    |   movel([0.182461, -1.429621, -2.539510, -0.743258, 1.570796, 1.753257],accel_mss,speed_ms,0,blend_radius_m)
    |   movel([0.183810, -1.429810, -2.539363, -0.743216, 1.570796, 1.754607],accel_mss,speed_ms,0,blend_radius_m)
    |   movel([0.185034, -1.430194, -2.539064, -0.743131, 1.570796, 1.755830],accel_mss,speed_ms,0,blend_radius_m)
    |   movel([0.186110, -1.430760, -2.538624, -0.743005, 1.570796, 1.756906],accel_mss,speed_ms,0,blend_radius_m)
    |   movel([0.187012, -1.431499, -2.538048, -0.742842, 1.570796, 1.757809],accel_mss,speed_ms,0,blend_radius_m)
    |   movel([0.187715, -1.432399, -2.537345, -0.742645, 1.570796, 1.758511],accel_mss,speed_ms,0,blend_radius_m)
    |   movel([0.188198, -1.433447, -2.536525, -0.742416, 1.570796, 1.758995],accel_mss,speed_ms,0,blend_radius_m)
    |   speed_ms = 0.005
    |   movel([0.188198, -1.425059, -2.532761, -0.754569, 1.570796, 1.758995],accel_mss,speed_ms,0,blend_radius_m)
    |   speed_ms = 0.040
    |   movel([0.160347, -1.408053, -2.545687, -0.758649, 1.570796, 1.731144],accel_mss,speed_ms,0,blend_radius_m)
    |   speed_ms = 0.005
    |   movel([0.160347, -1.416570, -2.549523, -0.746297, 1.570796, 1.731144],accel_mss,speed_ms,0,blend_radius_m)
    |   speed_ms = 0.025
    |   movel([0.161048, -1.416837, -2.549320, -0.746232, 1.570796, 1.731844],accel_mss,speed_ms,0,blend_radius_m)
    |   movel([0.161576, -1.417274, -2.548989, -0.746126, 1.570796, 1.732372],accel_mss,speed_ms,0,blend_radius_m)
    |   movel([0.161701, -1.417602, -2.548740, -0.746047, 1.570796, 1.732497],accel_mss,speed_ms,0,blend_radius_m)
    |   movel([0.161690, -1.417989, -2.548446, -0.745954, 1.570796, 1.732487],accel_mss,speed_ms,0,blend_radius_m)
    |   movel([0.161538, -1.418393, -2.548139, -0.745857, 1.570796, 1.732334],accel_mss,speed_ms,0,blend_radius_m)
    |   movel([0.161230, -1.418767, -2.547855, -0.745767, 1.570796, 1.732027],accel_mss,speed_ms,0,blend_radius_m)
    |   movel([0.160492, -1.419336, -2.547422, -0.745631, 1.570796, 1.731288],accel_mss,speed_ms,0,blend_radius_m)
    |   movel([0.160242, -1.419699, -2.547145, -0.745545, 1.570796, 1.731038],accel_mss,speed_ms,0,blend_radius_m)
    |   movel([0.160152, -1.420075, -2.546859, -0.745456, 1.570796, 1.730949],accel_mss,speed_ms,0,blend_radius_m)
    |   movel([0.160302, -1.420762, -2.546335, -0.745293, 1.570796, 1.731098],accel_mss,speed_ms,0,blend_radius_m)
    |   movel([0.160720, -1.421423, -2.545829, -0.745137, 1.570796, 1.731517],accel_mss,speed_ms,0,blend_radius_m)
    |   movel([0.161277, -1.421975, -2.545406, -0.745007, 1.570796, 1.732073],accel_mss,speed_ms,0,blend_radius_m)
    |   movel([0.161958, -1.422414, -2.545071, -0.744905, 1.570796, 1.732754],accel_mss,speed_ms,0,blend_radius_m)
    |   movel([0.162749, -1.422724, -2.544833, -0.744832, 1.570796, 1.733545],accel_mss,speed_ms,0,blend_radius_m)
    |   movel([0.162178, -1.423539, -2.544208, -0.744642, 1.570796, 1.732975],accel_mss,speed_ms,0,blend_radius_m)
    |   movel([0.161765, -1.424363, -2.543574, -0.744451, 1.570796, 1.732562],accel_mss,speed_ms,0,blend_radius_m)
    |   movel([0.161491, -1.425192, -2.542936, -0.744261, 1.570796, 1.732287],accel_mss,speed_ms,0,blend_radius_m)
    |   movel([0.161335, -1.426018, -2.542300, -0.744072, 1.570796, 1.732131],accel_mss,speed_ms,0,blend_radius_m)
    |   movel([0.161310, -1.427628, -2.541056, -0.743706, 1.570796, 1.732106],accel_mss,speed_ms,0,blend_radius_m)
    |   movel([0.161552, -1.429136, -2.539887, -0.743367, 1.570796, 1.732348],accel_mss,speed_ms,0,blend_radius_m)
    |   movel([0.161818, -1.430578, -2.538765, -0.743046, 1.570796, 1.732614],accel_mss,speed_ms,0,blend_radius_m)
    |   movel([0.161818, -1.431340, -2.538172, -0.742877, 1.570796, 1.732614],accel_mss,speed_ms,0,blend_radius_m)
    |   movel([0.161643, -1.432142, -2.537546, -0.742701, 1.570796, 1.732440],accel_mss,speed_ms,0,blend_radius_m)
    |   movel([0.161209, -1.432975, -2.536895, -0.742519, 1.570796, 1.732006],accel_mss,speed_ms,0,blend_radius_m)
    |   movel([0.160534, -1.433740, -2.536296, -0.742353, 1.570796, 1.731330],accel_mss,speed_ms,0,blend_radius_m)
    |   movel([0.159706, -1.434315, -2.535846, -0.742229, 1.570796, 1.730503],accel_mss,speed_ms,0,blend_radius_m)
    |   movel([0.158821, -1.434572, -2.535644, -0.742173, 1.570796, 1.729617],accel_mss,speed_ms,0,blend_radius_m)
    |   movel([0.159210, -1.435121, -2.535213, -0.742055, 1.570796, 1.730006],accel_mss,speed_ms,0,blend_radius_m)
    |   movel([0.159647, -1.436428, -2.534185, -0.741776, 1.570796, 1.730443],accel_mss,speed_ms,0,blend_radius_m)
    |   movel([0.159693, -1.437162, -2.533607, -0.741620, 1.570796, 1.730489],accel_mss,speed_ms,0,blend_radius_m)
    |   movel([0.159449, -1.438725, -2.532372, -0.741291, 1.570796, 1.730245],accel_mss,speed_ms,0,blend_radius_m)
    |   movel([0.159158, -1.439530, -2.531736, -0.741124, 1.570796, 1.729954],accel_mss,speed_ms,0,blend_radius_m)
    |   movel([0.158753, -1.440335, -2.531097, -0.740957, 1.570796, 1.729550],accel_mss,speed_ms,0,blend_radius_m)
    |   speed_ms = 0.005
    |   movel([0.158753, -1.432000, -2.527362, -0.753027, 1.570796, 1.729550],accel_mss,speed_ms,0,blend_radius_m)
    |   speed_ms = 0.040
    |   movel([0.154357, -1.432582, -2.526906, -0.752901, 1.570796, 1.725154],accel_mss,speed_ms,0,blend_radius_m)
    |   speed_ms = 0.005
    |   movel([0.154357, -1.440913, -2.530638, -0.740838, 1.570796, 1.725154],accel_mss,speed_ms,0,blend_radius_m)
    |   speed_ms = 0.025
    |   movel([0.157061, -1.447582, -2.525307, -0.739499, 1.570796, 1.727858],accel_mss,speed_ms,0,blend_radius_m)
    |   movel([0.157277, -1.448453, -2.524606, -0.739330, 1.570796, 1.728073],accel_mss,speed_ms,0,blend_radius_m)
    |   movel([0.157213, -1.448926, -2.524225, -0.739238, 1.570796, 1.728009],accel_mss,speed_ms,0,blend_radius_m)
    |   movel([0.156951, -1.449404, -2.523839, -0.739146, 1.570796, 1.727748],accel_mss,speed_ms,0,blend_radius_m)
    |   movel([0.156049, -1.450346, -2.523078, -0.738965, 1.570796, 1.726845],accel_mss,speed_ms,0,blend_radius_m)
    |   movel([0.155895, -1.450870, -2.522654, -0.738865, 1.570796, 1.726691],accel_mss,speed_ms,0,blend_radius_m)
    |   movel([0.155988, -1.451343, -2.522271, -0.738775, 1.570796, 1.726784],accel_mss,speed_ms,0,blend_radius_m)
    |   movel([0.156429, -1.451974, -2.521759, -0.738655, 1.570796, 1.727225],accel_mss,speed_ms,0,blend_radius_m)
    |   movel([0.157105, -1.452459, -2.521366, -0.738564, 1.570796, 1.727901],accel_mss,speed_ms,0,blend_radius_m)
    |   movel([0.158587, -1.453259, -2.520716, -0.738414, 1.570796, 1.729384],accel_mss,speed_ms,0,blend_radius_m)
    |   movel([0.159389, -1.453953, -2.520151, -0.738285, 1.570796, 1.730186],accel_mss,speed_ms,0,blend_radius_m)
    |   movel([0.160307, -1.455102, -2.519215, -0.738073, 1.570796, 1.731103],accel_mss,speed_ms,0,blend_radius_m)
    |   movel([0.160572, -1.455706, -2.518721, -0.737962, 1.570796, 1.731368],accel_mss,speed_ms,0,blend_radius_m)
    |   movel([0.160588, -1.456254, -2.518273, -0.737862, 1.570796, 1.731385],accel_mss,speed_ms,0,blend_radius_m)
    |   movel([0.160472, -1.456488, -2.518082, -0.737819, 1.570796, 1.731269],accel_mss,speed_ms,0,blend_radius_m)
    |   movel([0.160258, -1.456686, -2.517920, -0.737783, 1.570796, 1.731054],accel_mss,speed_ms,0,blend_radius_m)
    |   movel([0.159489, -1.456951, -2.517703, -0.737735, 1.570796, 1.730285],accel_mss,speed_ms,0,blend_radius_m)
    |   movel([0.159593, -1.457513, -2.517242, -0.737634, 1.570796, 1.730389],accel_mss,speed_ms,0,blend_radius_m)
    |   movel([0.159908, -1.458064, -2.516791, -0.737535, 1.570796, 1.730705],accel_mss,speed_ms,0,blend_radius_m)
    |   movel([0.160965, -1.459087, -2.515950, -0.737352, 1.570796, 1.731762],accel_mss,speed_ms,0,blend_radius_m)
    |   movel([0.163339, -1.460579, -2.514722, -0.737088, 1.570796, 1.734136],accel_mss,speed_ms,0,blend_radius_m)
    |   movel([0.164707, -1.461116, -2.514279, -0.736994, 1.570796, 1.735503],accel_mss,speed_ms,0,blend_radius_m)
    |   movel([0.166237, -1.461556, -2.513915, -0.736918, 1.570796, 1.737034],accel_mss,speed_ms,0,blend_radius_m)
    |   movel([0.167609, -1.462139, -2.513433, -0.736816, 1.570796, 1.738405],accel_mss,speed_ms,0,blend_radius_m)
    |   movel([0.168136, -1.462558, -2.513087, -0.736744, 1.570796, 1.738932],accel_mss,speed_ms,0,blend_radius_m)
    |   movel([0.168503, -1.463100, -2.512638, -0.736651, 1.570796, 1.739300],accel_mss,speed_ms,0,blend_radius_m)
    |   movel([0.168579, -1.463445, -2.512352, -0.736592, 1.570796, 1.739375],accel_mss,speed_ms,0,blend_radius_m)
    |   movel([0.168528, -1.463831, -2.512032, -0.736526, 1.570796, 1.739324],accel_mss,speed_ms,0,blend_radius_m)
    |   movel([0.168335, -1.464184, -2.511739, -0.736466, 1.570796, 1.739132],accel_mss,speed_ms,0,blend_radius_m)
    |   movel([0.167982, -1.464429, -2.511536, -0.736424, 1.570796, 1.738778],accel_mss,speed_ms,0,blend_radius_m)
    |   movel([0.167358, -1.464441, -2.511526, -0.736422, 1.570796, 1.738154],accel_mss,speed_ms,0,blend_radius_m)
    |   movel([0.164733, -1.463725, -2.512120, -0.736544, 1.570796, 1.735529],accel_mss,speed_ms,0,blend_radius_m)
    |   movel([0.162348, -1.462693, -2.512975, -0.736721, 1.570796, 1.733144],accel_mss,speed_ms,0,blend_radius_m)
    |   movel([0.162165, -1.463098, -2.512640, -0.736651, 1.570796, 1.732962],accel_mss,speed_ms,0,blend_radius_m)
    |   movel([0.162102, -1.463492, -2.512313, -0.736584, 1.570796, 1.732898],accel_mss,speed_ms,0,blend_radius_m)
    |   movel([0.162287, -1.464240, -2.511693, -0.736456, 1.570796, 1.733083],accel_mss,speed_ms,0,blend_radius_m)
    |   movel([0.162802, -1.464926, -2.511123, -0.736340, 1.570796, 1.733598],accel_mss,speed_ms,0,blend_radius_m)
    |   movel([0.163541, -1.465551, -2.510603, -0.736235, 1.570796, 1.734338],accel_mss,speed_ms,0,blend_radius_m)
    |   movel([0.165313, -1.466577, -2.509748, -0.736064, 1.570796, 1.736110],accel_mss,speed_ms,0,blend_radius_m)
    |   movel([0.166806, -1.467265, -2.509174, -0.735950, 1.570796, 1.737602],accel_mss,speed_ms,0,blend_radius_m)
    |   movel([0.167308, -1.467575, -2.508916, -0.735899, 1.570796, 1.738104],accel_mss,speed_ms,0,blend_radius_m)
    |   movel([0.167450, -1.467798, -2.508729, -0.735862, 1.570796, 1.738246],accel_mss,speed_ms,0,blend_radius_m)
    |   movel([0.167453, -1.468085, -2.508489, -0.735815, 1.570796, 1.738249],accel_mss,speed_ms,0,blend_radius_m)
    |   movel([0.167296, -1.468415, -2.508213, -0.735761, 1.570796, 1.738092],accel_mss,speed_ms,0,blend_radius_m)
    |   movel([0.167062, -1.468632, -2.508031, -0.735726, 1.570796, 1.737858],accel_mss,speed_ms,0,blend_radius_m)
    |   movel([0.166454, -1.468850, -2.507849, -0.735690, 1.570796, 1.737251],accel_mss,speed_ms,0,blend_radius_m)
    |   movel([0.165595, -1.469078, -2.507658, -0.735653, 1.570796, 1.736392],accel_mss,speed_ms,0,blend_radius_m)
    |   movel([0.165427, -1.469247, -2.507517, -0.735626, 1.570796, 1.736223],accel_mss,speed_ms,0,blend_radius_m)
    |   movel([0.165345, -1.469528, -2.507281, -0.735580, 1.570796, 1.736141],accel_mss,speed_ms,0,blend_radius_m)
    |   movel([0.165401, -1.469808, -2.507046, -0.735535, 1.570796, 1.736198],accel_mss,speed_ms,0,blend_radius_m)
    |   movel([0.165799, -1.470337, -2.506602, -0.735450, 1.570796, 1.736596],accel_mss,speed_ms,0,blend_radius_m)
    |   movel([0.166817, -1.471128, -2.505937, -0.735324, 1.570796, 1.737614],accel_mss,speed_ms,0,blend_radius_m)
    |   movel([0.171507, -1.474123, -2.503412, -0.734854, 1.570796, 1.742303],accel_mss,speed_ms,0,blend_radius_m)
    |   movel([0.171909, -1.474489, -2.503102, -0.734798, 1.570796, 1.742705],accel_mss,speed_ms,0,blend_radius_m)
    |   movel([0.172183, -1.474947, -2.502714, -0.734728, 1.570796, 1.742980],accel_mss,speed_ms,0,blend_radius_m)
    |   movel([0.172221, -1.475464, -2.502276, -0.734649, 1.570796, 1.743018],accel_mss,speed_ms,0,blend_radius_m)
    |   movel([0.171913, -1.476002, -2.501820, -0.734567, 1.570796, 1.742709],accel_mss,speed_ms,0,blend_radius_m)
    |   movel([0.171372, -1.476368, -2.501509, -0.734512, 1.570796, 1.742169],accel_mss,speed_ms,0,blend_radius_m)
    |   movel([0.170763, -1.476499, -2.501398, -0.734492, 1.570796, 1.741560],accel_mss,speed_ms,0,blend_radius_m)
    |   movel([0.170150, -1.476458, -2.501433, -0.734498, 1.570796, 1.740946],accel_mss,speed_ms,0,blend_radius_m)
    |   movel([0.169597, -1.476313, -2.501556, -0.734520, 1.570796, 1.740393],accel_mss,speed_ms,0,blend_radius_m)
    |   movel([0.166572, -1.475142, -2.502549, -0.734698, 1.570796, 1.737369],accel_mss,speed_ms,0,blend_radius_m)
    |   movel([0.163666, -1.473823, -2.503665, -0.734901, 1.570796, 1.734463],accel_mss,speed_ms,0,blend_radius_m)
    |   movel([0.160882, -1.472356, -2.504903, -0.735130, 1.570796, 1.731678],accel_mss,speed_ms,0,blend_radius_m)
    |   movel([0.158230, -1.470742, -2.506262, -0.735385, 1.570796, 1.729026],accel_mss,speed_ms,0,blend_radius_m)
    |   movel([0.157306, -1.470085, -2.506813, -0.735490, 1.570796, 1.728103],accel_mss,speed_ms,0,blend_radius_m)
    |   movel([0.156559, -1.469281, -2.507488, -0.735620, 1.570796, 1.727356],accel_mss,speed_ms,0,blend_radius_m)
    |   movel([0.156265, -1.468703, -2.507972, -0.735714, 1.570796, 1.727061],accel_mss,speed_ms,0,blend_radius_m)
    |   movel([0.156066, -1.468071, -2.508501, -0.735817, 1.570796, 1.726862],accel_mss,speed_ms,0,blend_radius_m)
    |   movel([0.155838, -1.466713, -2.509635, -0.736041, 1.570796, 1.726634],accel_mss,speed_ms,0,blend_radius_m)
    |   movel([0.155601, -1.461616, -2.513866, -0.736907, 1.570796, 1.726397],accel_mss,speed_ms,0,blend_radius_m)
    |   movel([0.155370, -1.460235, -2.515006, -0.737149, 1.570796, 1.726167],accel_mss,speed_ms,0,blend_radius_m)
    |   movel([0.154966, -1.459071, -2.515963, -0.737355, 1.570796, 1.725762],accel_mss,speed_ms,0,blend_radius_m)
    |   movel([0.154681, -1.458614, -2.516339, -0.737436, 1.570796, 1.725477],accel_mss,speed_ms,0,blend_radius_m)
    |   movel([0.154331, -1.458258, -2.516631, -0.737500, 1.570796, 1.725127],accel_mss,speed_ms,0,blend_radius_m)
    |   movel([0.153911, -1.458025, -2.516822, -0.737541, 1.570796, 1.724707],accel_mss,speed_ms,0,blend_radius_m)
    |   movel([0.153414, -1.457927, -2.516903, -0.737559, 1.570796, 1.724210],accel_mss,speed_ms,0,blend_radius_m)
    |   movel([0.152456, -1.457979, -2.516860, -0.737550, 1.570796, 1.723252],accel_mss,speed_ms,0,blend_radius_m)
    |   movel([0.152013, -1.457959, -2.516877, -0.737553, 1.570796, 1.722809],accel_mss,speed_ms,0,blend_radius_m)
    |   movel([0.151669, -1.457806, -2.517002, -0.737581, 1.570796, 1.722466],accel_mss,speed_ms,0,blend_radius_m)
    |   movel([0.151472, -1.457323, -2.517398, -0.737668, 1.570796, 1.722268],accel_mss,speed_ms,0,blend_radius_m)
    |   movel([0.151536, -1.456708, -2.517902, -0.737779, 1.570796, 1.722333],accel_mss,speed_ms,0,blend_radius_m)
    |   movel([0.151846, -1.454712, -2.519533, -0.738144, 1.570796, 1.722643],accel_mss,speed_ms,0,blend_radius_m)
    |   movel([0.152006, -1.452762, -2.521120, -0.738507, 1.570796, 1.722802],accel_mss,speed_ms,0,blend_radius_m)
    |   movel([0.151950, -1.448972, -2.524188, -0.739229, 1.570796, 1.722746],accel_mss,speed_ms,0,blend_radius_m)
    |   movel([0.151537, -1.445268, -2.527165, -0.739956, 1.570796, 1.722334],accel_mss,speed_ms,0,blend_radius_m)
    |   movel([0.150932, -1.441582, -2.530107, -0.740700, 1.570796, 1.721728],accel_mss,speed_ms,0,blend_radius_m)
    |   speed_ms = 0.005
    |   movel([0.150932, -1.433257, -2.526377, -0.752755, 1.570796, 1.721728],accel_mss,speed_ms,0,blend_radius_m)
    |   speed_ms = 0.040
    |   movel([0.148558, -1.439611, -2.521359, -0.751419, 1.570796, 1.719355],accel_mss,speed_ms,0,blend_radius_m)
    |   speed_ms = 0.005
    |   movel([0.148558, -1.447887, -2.525062, -0.739440, 1.570796, 1.719355],accel_mss,speed_ms,0,blend_radius_m)
    |   speed_ms = 0.025
    |   movel([0.147293, -1.452117, -2.521643, -0.738628, 1.570796, 1.718089],accel_mss,speed_ms,0,blend_radius_m)
    |   movel([0.146519, -1.454236, -2.519921, -0.738232, 1.570796, 1.717315],accel_mss,speed_ms,0,blend_radius_m)
    |   movel([0.145655, -1.456350, -2.518195, -0.737844, 1.570796, 1.716451],accel_mss,speed_ms,0,blend_radius_m)
    |   movel([0.144468, -1.455618, -2.518793, -0.737978, 1.570796, 1.715264],accel_mss,speed_ms,0,blend_radius_m)
    |   movel([0.144245, -1.455516, -2.518877, -0.737997, 1.570796, 1.715041],accel_mss,speed_ms,0,blend_radius_m)
    |   movel([0.143973, -1.455537, -2.518860, -0.737993, 1.570796, 1.714769],accel_mss,speed_ms,0,blend_radius_m)
    |   movel([0.143715, -1.455735, -2.518697, -0.737956, 1.570796, 1.714512],accel_mss,speed_ms,0,blend_radius_m)
    |   movel([0.143536, -1.456005, -2.518477, -0.737907, 1.570796, 1.714332],accel_mss,speed_ms,0,blend_radius_m)
    |   movel([0.142423, -1.457670, -2.517114, -0.737605, 1.570796, 1.713219],accel_mss,speed_ms,0,blend_radius_m)
    |   movel([0.141061, -1.459243, -2.515822, -0.737324, 1.570796, 1.711857],accel_mss,speed_ms,0,blend_radius_m)
    |   movel([0.140683, -1.459568, -2.515554, -0.737266, 1.570796, 1.711479],accel_mss,speed_ms,0,blend_radius_m)
    |   movel([0.140276, -1.459709, -2.515438, -0.737242, 1.570796, 1.711073],accel_mss,speed_ms,0,blend_radius_m)
    |   movel([0.140039, -1.459566, -2.515556, -0.737267, 1.570796, 1.710835],accel_mss,speed_ms,0,blend_radius_m)
    |   movel([0.139948, -1.459290, -2.515783, -0.737316, 1.570796, 1.710744],accel_mss,speed_ms,0,blend_radius_m)
    |   movel([0.139802, -1.457440, -2.517302, -0.737647, 1.570796, 1.710598],accel_mss,speed_ms,0,blend_radius_m)
    |   movel([0.140013, -1.455473, -2.518911, -0.738004, 1.570796, 1.710809],accel_mss,speed_ms,0,blend_radius_m)
    |   speed_ms = 0.005
    |   movel([0.140013, -1.447256, -2.515240, -0.749893, 1.570796, 1.710809],accel_mss,speed_ms,0,blend_radius_m)
    |   speed_ms = 0.040
    |   movel([0.143541, -1.450689, -2.512464, -0.749236, 1.570796, 1.714337],accel_mss,speed_ms,0,blend_radius_m)
    |   speed_ms = 0.005
    |   movel([0.143541, -1.458879, -2.516121, -0.737389, 1.570796, 1.714337],accel_mss,speed_ms,0,blend_radius_m)
    |   speed_ms = 0.025
    |   movel([0.143262, -1.461761, -2.513746, -0.736882, 1.570796, 1.714058],accel_mss,speed_ms,0,blend_radius_m)
    |   movel([0.142955, -1.463237, -2.512525, -0.736627, 1.570796, 1.713751],accel_mss,speed_ms,0,blend_radius_m)
    |   movel([0.142021, -1.466218, -2.510047, -0.736123, 1.570796, 1.712817],accel_mss,speed_ms,0,blend_radius_m)
    |   movel([0.141397, -1.467713, -2.508800, -0.735876, 1.570796, 1.712194],accel_mss,speed_ms,0,blend_radius_m)
    |   movel([0.139852, -1.470677, -2.506317, -0.735396, 1.570796, 1.710648],accel_mss,speed_ms,0,blend_radius_m)
    |   movel([0.140038, -1.469700, -2.507136, -0.735552, 1.570796, 1.710834],accel_mss,speed_ms,0,blend_radius_m)
    |   movel([0.139919, -1.468812, -2.507881, -0.735696, 1.570796, 1.710715],accel_mss,speed_ms,0,blend_radius_m)
    |   movel([0.139512, -1.468072, -2.508500, -0.735817, 1.570796, 1.710308],accel_mss,speed_ms,0,blend_radius_m)
    |   movel([0.138834, -1.467542, -2.508943, -0.735904, 1.570796, 1.709630],accel_mss,speed_ms,0,blend_radius_m)
    |   speed_ms = 0.005
    |   movel([0.138834, -1.459420, -2.505321, -0.747648, 1.570796, 1.709630],accel_mss,speed_ms,0,blend_radius_m)
    |   speed_ms = 0.040
    |   movel([0.126690, -1.463689, -2.501786, -0.746913, 1.570796, 1.697487],accel_mss,speed_ms,0,blend_radius_m)
    |   speed_ms = 0.005
    |   movel([0.126690, -1.471777, -2.505391, -0.735221, 1.570796, 1.697487],accel_mss,speed_ms,0,blend_radius_m)
    |   speed_ms = 0.025
    |   movel([0.124728, -1.473662, -2.503801, -0.734926, 1.570796, 1.695524],accel_mss,speed_ms,0,blend_radius_m)
    |   movel([0.122583, -1.475378, -2.502349, -0.734662, 1.570796, 1.693379],accel_mss,speed_ms,0,blend_radius_m)
    |   movel([0.120295, -1.476899, -2.501058, -0.734432, 1.570796, 1.691091],accel_mss,speed_ms,0,blend_radius_m)
    |   movel([0.117902, -1.478198, -2.499953, -0.734238, 1.570796, 1.688698],accel_mss,speed_ms,0,blend_radius_m)
    |   movel([0.118428, -1.477273, -2.500740, -0.734376, 1.570796, 1.689224],accel_mss,speed_ms,0,blend_radius_m)
    |   movel([0.118796, -1.476390, -2.501491, -0.734509, 1.570796, 1.689592],accel_mss,speed_ms,0,blend_radius_m)
    |   movel([0.118980, -1.475627, -2.502138, -0.734624, 1.570796, 1.689777],accel_mss,speed_ms,0,blend_radius_m)
    |   movel([0.118959, -1.475064, -2.502615, -0.734710, 1.570796, 1.689756],accel_mss,speed_ms,0,blend_radius_m)
    |   movel([0.118706, -1.474786, -2.502850, -0.734752, 1.570796, 1.689502],accel_mss,speed_ms,0,blend_radius_m)
    |   movel([0.118486, -1.474778, -2.502857, -0.734754, 1.570796, 1.689283],accel_mss,speed_ms,0,blend_radius_m)
    |   movel([0.118196, -1.474870, -2.502779, -0.734740, 1.570796, 1.688992],accel_mss,speed_ms,0,blend_radius_m)
    |   movel([0.117408, -1.475399, -2.502331, -0.734659, 1.570796, 1.688204],accel_mss,speed_ms,0,blend_radius_m)
    |   movel([0.115476, -1.477294, -2.500723, -0.734373, 1.570796, 1.686272],accel_mss,speed_ms,0,blend_radius_m)
    |   movel([0.114562, -1.478102, -2.500034, -0.734253, 1.570796, 1.685358],accel_mss,speed_ms,0,blend_radius_m)
    |   movel([0.112567, -1.479569, -2.498783, -0.734037, 1.570796, 1.683364],accel_mss,speed_ms,0,blend_radius_m)
    |   movel([0.111510, -1.480208, -2.498237, -0.733944, 1.570796, 1.682306],accel_mss,speed_ms,0,blend_radius_m)
    |   movel([0.110428, -1.480767, -2.497759, -0.733864, 1.570796, 1.681224],accel_mss,speed_ms,0,blend_radius_m)
    |   movel([0.109332, -1.481239, -2.497354, -0.733796, 1.570796, 1.680128],accel_mss,speed_ms,0,blend_radius_m)
    |   movel([0.108237, -1.481609, -2.497037, -0.733743, 1.570796, 1.679033],accel_mss,speed_ms,0,blend_radius_m)
    |   movel([0.109495, -1.480213, -2.498233, -0.733944, 1.570796, 1.680291],accel_mss,speed_ms,0,blend_radius_m)
    |   movel([0.110712, -1.478790, -2.499448, -0.734151, 1.570796, 1.681508],accel_mss,speed_ms,0,blend_radius_m)
    |   movel([0.111231, -1.477810, -2.500283, -0.734296, 1.570796, 1.682028],accel_mss,speed_ms,0,blend_radius_m)
    |   movel([0.111476, -1.476835, -2.501112, -0.734442, 1.570796, 1.682273],accel_mss,speed_ms,0,blend_radius_m)
    |   movel([0.111406, -1.476498, -2.501399, -0.734492, 1.570796, 1.682202],accel_mss,speed_ms,0,blend_radius_m)
    |   movel([0.111156, -1.476339, -2.501534, -0.734516, 1.570796, 1.681952],accel_mss,speed_ms,0,blend_radius_m)
    |   movel([0.110695, -1.476418, -2.501466, -0.734504, 1.570796, 1.681491],accel_mss,speed_ms,0,blend_radius_m)
    |   movel([0.109985, -1.476796, -2.501145, -0.734447, 1.570796, 1.680781],accel_mss,speed_ms,0,blend_radius_m)
    |   movel([0.106293, -1.479270, -2.499038, -0.734081, 1.570796, 1.677090],accel_mss,speed_ms,0,blend_radius_m)
    |   movel([0.104413, -1.480308, -2.498151, -0.733930, 1.570796, 1.675210],accel_mss,speed_ms,0,blend_radius_m)
    |   movel([0.103458, -1.480699, -2.497817, -0.733873, 1.570796, 1.674254],accel_mss,speed_ms,0,blend_radius_m)
    |   movel([0.102487, -1.480974, -2.497581, -0.733834, 1.570796, 1.673283],accel_mss,speed_ms,0,blend_radius_m)
    |   speed_ms = 0.005
    |   movel([0.102487, -1.472960, -2.494014, -0.745416, 1.570796, 1.673283],accel_mss,speed_ms,0,blend_radius_m)
    |   speed_ms = 0.040
    |   movel([0.118652, -1.454320, -2.509507, -0.748562, 1.570796, 1.689448],accel_mss,speed_ms,0,blend_radius_m)
    |   speed_ms = 0.005
    |   movel([0.118652, -1.462482, -2.513150, -0.736757, 1.570796, 1.689448],accel_mss,speed_ms,0,blend_radius_m)
    |   speed_ms = 0.025
    |   movel([0.118575, -1.461266, -2.514155, -0.736968, 1.570796, 1.689372],accel_mss,speed_ms,0,blend_radius_m)
    |   movel([0.118788, -1.459980, -2.515216, -0.737194, 1.570796, 1.689584],accel_mss,speed_ms,0,blend_radius_m)
    |   movel([0.119258, -1.458648, -2.516311, -0.737430, 1.570796, 1.690055],accel_mss,speed_ms,0,blend_radius_m)
    |   movel([0.119955, -1.457301, -2.517416, -0.737672, 1.570796, 1.690752],accel_mss,speed_ms,0,blend_radius_m)
    |   movel([0.120854, -1.455963, -2.518511, -0.737915, 1.570796, 1.691651],accel_mss,speed_ms,0,blend_radius_m)
    |   movel([0.121920, -1.454666, -2.519570, -0.738153, 1.570796, 1.692717],accel_mss,speed_ms,0,blend_radius_m)
    |   movel([0.123128, -1.453435, -2.520573, -0.738381, 1.570796, 1.693924],accel_mss,speed_ms,0,blend_radius_m)
    |   movel([0.124442, -1.452300, -2.521495, -0.738594, 1.570796, 1.695239],accel_mss,speed_ms,0,blend_radius_m)
    |   movel([0.126164, -1.451030, -2.522525, -0.738834, 1.570796, 1.696960],accel_mss,speed_ms,0,blend_radius_m)
    |   movel([0.129687, -1.448583, -2.524501, -0.739304, 1.570796, 1.700483],accel_mss,speed_ms,0,blend_radius_m)
    |   movel([0.131359, -1.447249, -2.525575, -0.739565, 1.570796, 1.702155],accel_mss,speed_ms,0,blend_radius_m)
    |   movel([0.132860, -1.445714, -2.526807, -0.739867, 1.570796, 1.703657],accel_mss,speed_ms,0,blend_radius_m)
    |   movel([0.133496, -1.444883, -2.527473, -0.740033, 1.570796, 1.704293],accel_mss,speed_ms,0,blend_radius_m)
    |   movel([0.134024, -1.444034, -2.528152, -0.740203, 1.570796, 1.704821],accel_mss,speed_ms,0,blend_radius_m)
    |   movel([0.134421, -1.443187, -2.528828, -0.740374, 1.570796, 1.705217],accel_mss,speed_ms,0,blend_radius_m)
    |   movel([0.134665, -1.442360, -2.529488, -0.740542, 1.570796, 1.705461],accel_mss,speed_ms,0,blend_radius_m)
    |   movel([0.134728, -1.441575, -2.530112, -0.740702, 1.570796, 1.705524],accel_mss,speed_ms,0,blend_radius_m)
    |   movel([0.134585, -1.440854, -2.530685, -0.740850, 1.570796, 1.705381],accel_mss,speed_ms,0,blend_radius_m)
    |   speed_ms = 0.005
    |   movel([0.134585, -1.432523, -2.526953, -0.752914, 1.570796, 1.705381],accel_mss,speed_ms,0,blend_radius_m)
    |   speed_ms = 0.040
    |   movel([0.133004, -1.426801, -2.531413, -0.754175, 1.570796, 1.703800],accel_mss,speed_ms,0,blend_radius_m)
    |   speed_ms = 0.005
    |   movel([0.133004, -1.435175, -2.535170, -0.742043, 1.570796, 1.703800],accel_mss,speed_ms,0,blend_radius_m)
    |   speed_ms = 0.025
    |   movel([0.131954, -1.439890, -2.531450, -0.741049, 1.570796, 1.702750],accel_mss,speed_ms,0,blend_radius_m)
    |   movel([0.131474, -1.440949, -2.530610, -0.740830, 1.570796, 1.702271],accel_mss,speed_ms,0,blend_radius_m)
    |   movel([0.130669, -1.441933, -2.529828, -0.740629, 1.570796, 1.701465],accel_mss,speed_ms,0,blend_radius_m)
    |   movel([0.129641, -1.442790, -2.529145, -0.740454, 1.570796, 1.700437],accel_mss,speed_ms,0,blend_radius_m)
    |   movel([0.126104, -1.445221, -2.527202, -0.739965, 1.570796, 1.696900],accel_mss,speed_ms,0,blend_radius_m)
    |   movel([0.124928, -1.446193, -2.526423, -0.739773, 1.570796, 1.695724],accel_mss,speed_ms,0,blend_radius_m)
    |   movel([0.123829, -1.447231, -2.525590, -0.739568, 1.570796, 1.694626],accel_mss,speed_ms,0,blend_radius_m)
    |   movel([0.122817, -1.448321, -2.524713, -0.739355, 1.570796, 1.693613],accel_mss,speed_ms,0,blend_radius_m)
    |   movel([0.121989, -1.449445, -2.523806, -0.739138, 1.570796, 1.692785],accel_mss,speed_ms,0,blend_radius_m)
    |   movel([0.121311, -1.450605, -2.522869, -0.738915, 1.570796, 1.692107],accel_mss,speed_ms,0,blend_radius_m)
    |   movel([0.120646, -1.451760, -2.521933, -0.738696, 1.570796, 1.691443],accel_mss,speed_ms,0,blend_radius_m)
    |   movel([0.119860, -1.452874, -2.521028, -0.738486, 1.570796, 1.690656],accel_mss,speed_ms,0,blend_radius_m)
    |   movel([0.118748, -1.450438, -2.523003, -0.738947, 1.570796, 1.689544],accel_mss,speed_ms,0,blend_radius_m)
    |   movel([0.118765, -1.449672, -2.523623, -0.739094, 1.570796, 1.689562],accel_mss,speed_ms,0,blend_radius_m)
    |   movel([0.118930, -1.448892, -2.524253, -0.739245, 1.570796, 1.689726],accel_mss,speed_ms,0,blend_radius_m)
    |   movel([0.119240, -1.448096, -2.524894, -0.739399, 1.570796, 1.690036],accel_mss,speed_ms,0,blend_radius_m)
    |   movel([0.119703, -1.447279, -2.525552, -0.739559, 1.570796, 1.690499],accel_mss,speed_ms,0,blend_radius_m)
    |   movel([0.120629, -1.446199, -2.526419, -0.739771, 1.570796, 1.691425],accel_mss,speed_ms,0,blend_radius_m)
    |   movel([0.122024, -1.444944, -2.527424, -0.740021, 1.570796, 1.692820],accel_mss,speed_ms,0,blend_radius_m)
    |   movel([0.125487, -1.442187, -2.529625, -0.740577, 1.570796, 1.696284],accel_mss,speed_ms,0,blend_radius_m)
    |   movel([0.127192, -1.440827, -2.530706, -0.740855, 1.570796, 1.697988],accel_mss,speed_ms,0,blend_radius_m)
    |   movel([0.128630, -1.439573, -2.531701, -0.741115, 1.570796, 1.699426],accel_mss,speed_ms,0,blend_radius_m)
    |   movel([0.129616, -1.438498, -2.532552, -0.741339, 1.570796, 1.700412],accel_mss,speed_ms,0,blend_radius_m)
    |   movel([0.129882, -1.438049, -2.532907, -0.741433, 1.570796, 1.700679],accel_mss,speed_ms,0,blend_radius_m)
    |   movel([0.129964, -1.437670, -2.533206, -0.741513, 1.570796, 1.700761],accel_mss,speed_ms,0,blend_radius_m)
    |   speed_ms = 0.005
    |   movel([0.129964, -1.429314, -2.529460, -0.753615, 1.570796, 1.700761],accel_mss,speed_ms,0,blend_radius_m)
    |   speed_ms = 0.040
    |   movel([0.122893, -1.428717, -2.529925, -0.753747, 1.570796, 1.693690],accel_mss,speed_ms,0,blend_radius_m)
    |   speed_ms = 0.005
    |   movel([0.122893, -1.437077, -2.533674, -0.741638, 1.570796, 1.693690],accel_mss,speed_ms,0,blend_radius_m)
    |   speed_ms = 0.025
    |   movel([0.122209, -1.437007, -2.533729, -0.741653, 1.570796, 1.693006],accel_mss,speed_ms,0,blend_radius_m)
    |   movel([0.121626, -1.436800, -2.533892, -0.741697, 1.570796, 1.692422],accel_mss,speed_ms,0,blend_radius_m)
    |   movel([0.120719, -1.436071, -2.534466, -0.741852, 1.570796, 1.691516],accel_mss,speed_ms,0,blend_radius_m)
    |   movel([0.120087, -1.435054, -2.535266, -0.742070, 1.570796, 1.690884],accel_mss,speed_ms,0,blend_radius_m)
    |   movel([0.119648, -1.433912, -2.536162, -0.742316, 1.570796, 1.690444],accel_mss,speed_ms,0,blend_radius_m)
    |   movel([0.119577, -1.433458, -2.536517, -0.742414, 1.570796, 1.690374],accel_mss,speed_ms,0,blend_radius_m)
    |   movel([0.119940, -1.432671, -2.537133, -0.742585, 1.570796, 1.690736],accel_mss,speed_ms,0,blend_radius_m)
    |   movel([0.121281, -1.430471, -2.538849, -0.743069, 1.570796, 1.692078],accel_mss,speed_ms,0,blend_radius_m)
    |   movel([0.123710, -1.426009, -2.542307, -0.744074, 1.570796, 1.694506],accel_mss,speed_ms,0,blend_radius_m)
    |   movel([0.124792, -1.423757, -2.544040, -0.744592, 1.570796, 1.695589],accel_mss,speed_ms,0,blend_radius_m)
    |   speed_ms = 0.005
    |   movel([0.124792, -1.415295, -2.540235, -0.756859, 1.570796, 1.695589],accel_mss,speed_ms,0,blend_radius_m)
    |   speed_ms = 0.040
    |   movel([0.120439, -1.416998, -2.538942, -0.756450, 1.570796, 1.691236],accel_mss,speed_ms,0,blend_radius_m)
    |   speed_ms = 0.005
    |   movel([0.120439, -1.425447, -2.542740, -0.744202, 1.570796, 1.691236],accel_mss,speed_ms,0,blend_radius_m)
    |   speed_ms = 0.025
    |   movel([0.119935, -1.426809, -2.541688, -0.743891, 1.570796, 1.690731],accel_mss,speed_ms,0,blend_radius_m)
    |   movel([0.119253, -1.428166, -2.540638, -0.743584, 1.570796, 1.690049],accel_mss,speed_ms,0,blend_radius_m)
    |   movel([0.118343, -1.429439, -2.539651, -0.743299, 1.570796, 1.689139],accel_mss,speed_ms,0,blend_radius_m)
    |   movel([0.117785, -1.430022, -2.539198, -0.743169, 1.570796, 1.688582],accel_mss,speed_ms,0,blend_radius_m)
    |   movel([0.116540, -1.431083, -2.538372, -0.742934, 1.570796, 1.687336],accel_mss,speed_ms,0,blend_radius_m)
    |   movel([0.116272, -1.431628, -2.537947, -0.742814, 1.570796, 1.687068],accel_mss,speed_ms,0,blend_radius_m)
    |   movel([0.114788, -1.435842, -2.534646, -0.741901, 1.570796, 1.685584],accel_mss,speed_ms,0,blend_radius_m)
    |   movel([0.114658, -1.436249, -2.534326, -0.741814, 1.570796, 1.685455],accel_mss,speed_ms,0,blend_radius_m)
    |   movel([0.114654, -1.436620, -2.534034, -0.741735, 1.570796, 1.685450],accel_mss,speed_ms,0,blend_radius_m)
    |   movel([0.114992, -1.436970, -2.533758, -0.741661, 1.570796, 1.685789],accel_mss,speed_ms,0,blend_radius_m)
    |   movel([0.115542, -1.437129, -2.533633, -0.741627, 1.570796, 1.686338],accel_mss,speed_ms,0,blend_radius_m)
    |   movel([0.117152, -1.437524, -2.533321, -0.741544, 1.570796, 1.687949],accel_mss,speed_ms,0,blend_radius_m)
    |   movel([0.118641, -1.438082, -2.532881, -0.741426, 1.570796, 1.689437],accel_mss,speed_ms,0,blend_radius_m)
    |   movel([0.119908, -1.438862, -2.532264, -0.741263, 1.570796, 1.690705],accel_mss,speed_ms,0,blend_radius_m)
    |   movel([0.120845, -1.439931, -2.531417, -0.741040, 1.570796, 1.691642],accel_mss,speed_ms,0,blend_radius_m)
    |   speed_ms = 0.005
    |   movel([0.120845, -1.431593, -2.527681, -0.753115, 1.570796, 1.691642],accel_mss,speed_ms,0,blend_radius_m)
    |   speed_ms = 0.040
    |   movel([0.117067, -1.442493, -2.519063, -0.750834, 1.570796, 1.687863],accel_mss,speed_ms,0,blend_radius_m)
    |   speed_ms = 0.005
    |   movel([0.117067, -1.450747, -2.522754, -0.738888, 1.570796, 1.687863],accel_mss,speed_ms,0,blend_radius_m)
    |   speed_ms = 0.025
    |   movel([0.116755, -1.450955, -2.522585, -0.738849, 1.570796, 1.687552],accel_mss,speed_ms,0,blend_radius_m)
    |   movel([0.116482, -1.451240, -2.522354, -0.738794, 1.570796, 1.687279],accel_mss,speed_ms,0,blend_radius_m)
    |   movel([0.115440, -1.452783, -2.521102, -0.738503, 1.570796, 1.686236],accel_mss,speed_ms,0,blend_radius_m)
    |   movel([0.115251, -1.452911, -2.520998, -0.738479, 1.570796, 1.686047],accel_mss,speed_ms,0,blend_radius_m)
    |   movel([0.114957, -1.452931, -2.520983, -0.738476, 1.570796, 1.685753],accel_mss,speed_ms,0,blend_radius_m)
    |   movel([0.114717, -1.452784, -2.521102, -0.738503, 1.570796, 1.685513],accel_mss,speed_ms,0,blend_radius_m)
    |   movel([0.114388, -1.452168, -2.521602, -0.738619, 1.570796, 1.685184],accel_mss,speed_ms,0,blend_radius_m)
    |   movel([0.114191, -1.450864, -2.522659, -0.738866, 1.570796, 1.684987],accel_mss,speed_ms,0,blend_radius_m)
    |   movel([0.114441, -1.449533, -2.523735, -0.739121, 1.570796, 1.685237],accel_mss,speed_ms,0,blend_radius_m)
    |   movel([0.114918, -1.448160, -2.524842, -0.739387, 1.570796, 1.685715],accel_mss,speed_ms,0,blend_radius_m)
    |   movel([0.115514, -1.446802, -2.525935, -0.739652, 1.570796, 1.686310],accel_mss,speed_ms,0,blend_radius_m)
    |   movel([0.116247, -1.445501, -2.526978, -0.739910, 1.570796, 1.687043],accel_mss,speed_ms,0,blend_radius_m)
    |   movel([0.117110, -1.444258, -2.527973, -0.740158, 1.570796, 1.687906],accel_mss,speed_ms,0,blend_radius_m)
    |   movel([0.118098, -1.443071, -2.528921, -0.740397, 1.570796, 1.688895],accel_mss,speed_ms,0,blend_radius_m)
    |   movel([0.119208, -1.441937, -2.529825, -0.740628, 1.570796, 1.690004],accel_mss,speed_ms,0,blend_radius_m)
    |   movel([0.120429, -1.440856, -2.530683, -0.740849, 1.570796, 1.691225],accel_mss,speed_ms,0,blend_radius_m)
    |   movel([0.121760, -1.439825, -2.531502, -0.741063, 1.570796, 1.692556],accel_mss,speed_ms,0,blend_radius_m)
    |   movel([0.123193, -1.438843, -2.532279, -0.741267, 1.570796, 1.693989],accel_mss,speed_ms,0,blend_radius_m)
    |   movel([0.125150, -1.437339, -2.533467, -0.741583, 1.570796, 1.695946],accel_mss,speed_ms,0,blend_radius_m)
    |   movel([0.127154, -1.435515, -2.534903, -0.741971, 1.570796, 1.697951],accel_mss,speed_ms,0,blend_radius_m)
    |   movel([0.129283, -1.433367, -2.536588, -0.742434, 1.570796, 1.700079],accel_mss,speed_ms,0,blend_radius_m)
    |   speed_ms = 0.005
    |   movel([0.129283, -1.424978, -2.532824, -0.754587, 1.570796, 1.700079],accel_mss,speed_ms,0,blend_radius_m)
    |   speed_ms = 0.040
    |   movel([0.127232, -1.425091, -2.532736, -0.754561, 1.570796, 1.698028],accel_mss,speed_ms,0,blend_radius_m)
    |   speed_ms = 0.005
    |   movel([0.127232, -1.433479, -2.536500, -0.742409, 1.570796, 1.698028],accel_mss,speed_ms,0,blend_radius_m)
    |   speed_ms = 0.025
    |   movel([0.128714, -1.430246, -2.539024, -0.743119, 1.570796, 1.699510],accel_mss,speed_ms,0,blend_radius_m)
    |   movel([0.130407, -1.427011, -2.541533, -0.743845, 1.570796, 1.701204],accel_mss,speed_ms,0,blend_radius_m)
    |   movel([0.131385, -1.425421, -2.542760, -0.744208, 1.570796, 1.702181],accel_mss,speed_ms,0,blend_radius_m)
    |   movel([0.132470, -1.423864, -2.543958, -0.744567, 1.570796, 1.703266],accel_mss,speed_ms,0,blend_radius_m)
    |   movel([0.133689, -1.422351, -2.545118, -0.744919, 1.570796, 1.704486],accel_mss,speed_ms,0,blend_radius_m)
    |   movel([0.135054, -1.420898, -2.546230, -0.745261, 1.570796, 1.705850],accel_mss,speed_ms,0,blend_radius_m)
    |   movel([0.138900, -1.417385, -2.548904, -0.746099, 1.570796, 1.709697],accel_mss,speed_ms,0,blend_radius_m)
    |   movel([0.140533, -1.415752, -2.550142, -0.746496, 1.570796, 1.711330],accel_mss,speed_ms,0,blend_radius_m)
    |   movel([0.141287, -1.414895, -2.550789, -0.746705, 1.570796, 1.712083],accel_mss,speed_ms,0,blend_radius_m)
    |   movel([0.141949, -1.413997, -2.551466, -0.746926, 1.570796, 1.712745],accel_mss,speed_ms,0,blend_radius_m)
    |   movel([0.143293, -1.411156, -2.553601, -0.747632, 1.570796, 1.714090],accel_mss,speed_ms,0,blend_radius_m)
    |   speed_ms = 0.005
    |   movel([0.143293, -1.402599, -2.549742, -0.760049, 1.570796, 1.714090],accel_mss,speed_ms,0,blend_radius_m)
    |   speed_ms = 0.040
    |   movel([0.146560, -1.395993, -2.554595, -0.761802, 1.570796, 1.717356],accel_mss,speed_ms,0,blend_radius_m)
    |   speed_ms = 0.005
    |   movel([0.146560, -1.404599, -2.558482, -0.749308, 1.570796, 1.717356],accel_mss,speed_ms,0,blend_radius_m)
    |   speed_ms = 0.025
    |   movel([0.147542, -1.402261, -2.560207, -0.749921, 1.570796, 1.718338],accel_mss,speed_ms,0,blend_radius_m)
    |   movel([0.148254, -1.401140, -2.561032, -0.750217, 1.570796, 1.719050],accel_mss,speed_ms,0,blend_radius_m)
    |   movel([0.149204, -1.400114, -2.561785, -0.750491, 1.570796, 1.720001],accel_mss,speed_ms,0,blend_radius_m)
    |   movel([0.150010, -1.399501, -2.562233, -0.750655, 1.570796, 1.720807],accel_mss,speed_ms,0,blend_radius_m)
    |   movel([0.150876, -1.398984, -2.562612, -0.750793, 1.570796, 1.721672],accel_mss,speed_ms,0,blend_radius_m)
    |   movel([0.152682, -1.398093, -2.563263, -0.751033, 1.570796, 1.723478],accel_mss,speed_ms,0,blend_radius_m)
    |   movel([0.154275, -1.397175, -2.563932, -0.751282, 1.570796, 1.725072],accel_mss,speed_ms,0,blend_radius_m)
    |   movel([0.155504, -1.396165, -2.564668, -0.751557, 1.570796, 1.726301],accel_mss,speed_ms,0,blend_radius_m)
    |   movel([0.157746, -1.393658, -2.566486, -0.752245, 1.570796, 1.728542],accel_mss,speed_ms,0,blend_radius_m)
    |   movel([0.158241, -1.393174, -2.566836, -0.752379, 1.570796, 1.729037],accel_mss,speed_ms,0,blend_radius_m)
    |   movel([0.158800, -1.392767, -2.567130, -0.752492, 1.570796, 1.729596],accel_mss,speed_ms,0,blend_radius_m)
    |   movel([0.160053, -1.392123, -2.567595, -0.752671, 1.570796, 1.730850],accel_mss,speed_ms,0,blend_radius_m)
    |   movel([0.162647, -1.391053, -2.568365, -0.752970, 1.570796, 1.733443],accel_mss,speed_ms,0,blend_radius_m)
    |   movel([0.165341, -1.389680, -2.569353, -0.753357, 1.570796, 1.736138],accel_mss,speed_ms,0,blend_radius_m)
    |   movel([0.166652, -1.388882, -2.569925, -0.753583, 1.570796, 1.737448],accel_mss,speed_ms,0,blend_radius_m)
    |   movel([0.167889, -1.387947, -2.570594, -0.753848, 1.570796, 1.738685],accel_mss,speed_ms,0,blend_radius_m)
    |   movel([0.168754, -1.387045, -2.571238, -0.754106, 1.570796, 1.739550],accel_mss,speed_ms,0,blend_radius_m)
    |   movel([0.169381, -1.386053, -2.571946, -0.754390, 1.570796, 1.740177],accel_mss,speed_ms,0,blend_radius_m)
    |   movel([0.169606, -1.385140, -2.572595, -0.754653, 1.570796, 1.740403],accel_mss,speed_ms,0,blend_radius_m)
    |   movel([0.169519, -1.384770, -2.572859, -0.754761, 1.570796, 1.740315],accel_mss,speed_ms,0,blend_radius_m)
    |   movel([0.169270, -1.384485, -2.573061, -0.754843, 1.570796, 1.740066],accel_mss,speed_ms,0,blend_radius_m)
    |   movel([0.168479, -1.384144, -2.573303, -0.754942, 1.570796, 1.739275],accel_mss,speed_ms,0,blend_radius_m)
    |   movel([0.167442, -1.384003, -2.573403, -0.754983, 1.570796, 1.738238],accel_mss,speed_ms,0,blend_radius_m)
    |   movel([0.166225, -1.384046, -2.573372, -0.754970, 1.570796, 1.737021],accel_mss,speed_ms,0,blend_radius_m)
    |   movel([0.164906, -1.384249, -2.573229, -0.754912, 1.570796, 1.735702],accel_mss,speed_ms,0,blend_radius_m)
    |   movel([0.163556, -1.384597, -2.572982, -0.754811, 1.570796, 1.734352],accel_mss,speed_ms,0,blend_radius_m)
    |   movel([0.162248, -1.385064, -2.572649, -0.754675, 1.570796, 1.733044],accel_mss,speed_ms,0,blend_radius_m)
    |   movel([0.161055, -1.385635, -2.572243, -0.754511, 1.570796, 1.731852],accel_mss,speed_ms,0,blend_radius_m)
    |   movel([0.160048, -1.386288, -2.571778, -0.754323, 1.570796, 1.730844],accel_mss,speed_ms,0,blend_radius_m)
    |   movel([0.158742, -1.387494, -2.570918, -0.753977, 1.570796, 1.729539],accel_mss,speed_ms,0,blend_radius_m)
    |   movel([0.155183, -1.391346, -2.568154, -0.752888, 1.570796, 1.725979],accel_mss,speed_ms,0,blend_radius_m)
    |   movel([0.152633, -1.393765, -2.566408, -0.752216, 1.570796, 1.723429],accel_mss,speed_ms,0,blend_radius_m)
    |   movel([0.150210, -1.395629, -2.565057, -0.751703, 1.570796, 1.721006],accel_mss,speed_ms,0,blend_radius_m)
    |   movel([0.148999, -1.396527, -2.564404, -0.751458, 1.570796, 1.719795],accel_mss,speed_ms,0,blend_radius_m)
    |   movel([0.147874, -1.397498, -2.563696, -0.751194, 1.570796, 1.718670],accel_mss,speed_ms,0,blend_radius_m)
    |   movel([0.146843, -1.398606, -2.562888, -0.750895, 1.570796, 1.717640],accel_mss,speed_ms,0,blend_radius_m)
    |   movel([0.145945, -1.399759, -2.562045, -0.750586, 1.570796, 1.716741],accel_mss,speed_ms,0,blend_radius_m)
    |   movel([0.145164, -1.400949, -2.561172, -0.750268, 1.570796, 1.715961],accel_mss,speed_ms,0,blend_radius_m)
    |   movel([0.144485, -1.402160, -2.560281, -0.749947, 1.570796, 1.715281],accel_mss,speed_ms,0,blend_radius_m)
    |   movel([0.143361, -1.404609, -2.558475, -0.749305, 1.570796, 1.714158],accel_mss,speed_ms,0,blend_radius_m)
    |   movel([0.142436, -1.407016, -2.556691, -0.748683, 1.570796, 1.713232],accel_mss,speed_ms,0,blend_radius_m)
    |   speed_ms = 0.005
    |   movel([0.142436, -1.398427, -2.552813, -0.761148, 1.570796, 1.713232],accel_mss,speed_ms,0,blend_radius_m)
    |   speed_ms = 0.040
    |   movel([0.139149, -1.400176, -2.551529, -0.760684, 1.570796, 1.709945],accel_mss,speed_ms,0,blend_radius_m)
    |   speed_ms = 0.005
    |   movel([0.139149, -1.408751, -2.555398, -0.748239, 1.570796, 1.709945],accel_mss,speed_ms,0,blend_radius_m)
    |   speed_ms = 0.025
    |   movel([0.140740, -1.404959, -2.558216, -0.749214, 1.570796, 1.711537],accel_mss,speed_ms,0,blend_radius_m)
    |   movel([0.141482, -1.403375, -2.559387, -0.749628, 1.570796, 1.712278],accel_mss,speed_ms,0,blend_radius_m)
    |   movel([0.142125, -1.401789, -2.560554, -0.750045, 1.570796, 1.712921],accel_mss,speed_ms,0,blend_radius_m)
    |   movel([0.142487, -1.400435, -2.561549, -0.750405, 1.570796, 1.713284],accel_mss,speed_ms,0,blend_radius_m)
    |   movel([0.142642, -1.399121, -2.562511, -0.750756, 1.570796, 1.713438],accel_mss,speed_ms,0,blend_radius_m)
    |   movel([0.142586, -1.397873, -2.563423, -0.751093, 1.570796, 1.713382],accel_mss,speed_ms,0,blend_radius_m)
    |   movel([0.142318, -1.396719, -2.564265, -0.751406, 1.570796, 1.713114],accel_mss,speed_ms,0,blend_radius_m)
    |   movel([0.142998, -1.396438, -2.564469, -0.751482, 1.570796, 1.713794],accel_mss,speed_ms,0,blend_radius_m)
    |   movel([0.143677, -1.396296, -2.564572, -0.751521, 1.570796, 1.714473],accel_mss,speed_ms,0,blend_radius_m)
    |   movel([0.145020, -1.396183, -2.564654, -0.751552, 1.570796, 1.715816],accel_mss,speed_ms,0,blend_radius_m)
    |   movel([0.146419, -1.395958, -2.564818, -0.751613, 1.570796, 1.717215],accel_mss,speed_ms,0,blend_radius_m)
    |   movel([0.147105, -1.395692, -2.565011, -0.751686, 1.570796, 1.717901],accel_mss,speed_ms,0,blend_radius_m)
    |   movel([0.147724, -1.395259, -2.565325, -0.751804, 1.570796, 1.718521],accel_mss,speed_ms,0,blend_radius_m)
    |   movel([0.154452, -1.389208, -2.569691, -0.753490, 1.570796, 1.725248],accel_mss,speed_ms,0,blend_radius_m)
    |   movel([0.154365, -1.388357, -2.570301, -0.753732, 1.570796, 1.725162],accel_mss,speed_ms,0,blend_radius_m)
    |   movel([0.153978, -1.387633, -2.570819, -0.753938, 1.570796, 1.724774],accel_mss,speed_ms,0,blend_radius_m)
    |   movel([0.153312, -1.387073, -2.571218, -0.754098, 1.570796, 1.724108],accel_mss,speed_ms,0,blend_radius_m)
    |   movel([0.152398, -1.386715, -2.571474, -0.754200, 1.570796, 1.723194],accel_mss,speed_ms,0,blend_radius_m)
    |   movel([0.153985, -1.386326, -2.571751, -0.754312, 1.570796, 1.724781],accel_mss,speed_ms,0,blend_radius_m)
    |   movel([0.155496, -1.386196, -2.571844, -0.754349, 1.570796, 1.726292],accel_mss,speed_ms,0,blend_radius_m)
    |   movel([0.156853, -1.386325, -2.571752, -0.754312, 1.570796, 1.727649],accel_mss,speed_ms,0,blend_radius_m)
    |   movel([0.157984, -1.386713, -2.571475, -0.754201, 1.570796, 1.728781],accel_mss,speed_ms,0,blend_radius_m)
    |   speed_ms = 0.005
    |   movel([0.157984, -1.377976, -2.567510, -0.766903, 1.570796, 1.728781],accel_mss,speed_ms,0,blend_radius_m)
    |   speed_ms = 0.040
    |   movel([0.158689, -1.374499, -2.569948, -0.767941, 1.570796, 1.729485],accel_mss,speed_ms,0,blend_radius_m)
    |   speed_ms = 0.005
    |   movel([0.158689, -1.383262, -2.573929, -0.755199, 1.570796, 1.729485],accel_mss,speed_ms,0,blend_radius_m)
    |   speed_ms = 0.025
    |   movel([0.159378, -1.381417, -2.575233, -0.755739, 1.570796, 1.730175],accel_mss,speed_ms,0,blend_radius_m)
    |   movel([0.159876, -1.379662, -2.576469, -0.756258, 1.570796, 1.730673],accel_mss,speed_ms,0,blend_radius_m)
    |   movel([0.160196, -1.377984, -2.577647, -0.756758, 1.570796, 1.730993],accel_mss,speed_ms,0,blend_radius_m)
    |   movel([0.160349, -1.376371, -2.578775, -0.757243, 1.570796, 1.731145],accel_mss,speed_ms,0,blend_radius_m)
    |   movel([0.160346, -1.374807, -2.579866, -0.757716, 1.570796, 1.731142],accel_mss,speed_ms,0,blend_radius_m)
    |   movel([0.160198, -1.373278, -2.580928, -0.758182, 1.570796, 1.730994],accel_mss,speed_ms,0,blend_radius_m)
    |   movel([0.159519, -1.370269, -2.583011, -0.759110, 1.570796, 1.730315],accel_mss,speed_ms,0,blend_radius_m)
    |   movel([0.157317, -1.376600, -2.578616, -0.757174, 1.570796, 1.728113],accel_mss,speed_ms,0,blend_radius_m)
    |   movel([0.157486, -1.375906, -2.579100, -0.757383, 1.570796, 1.728283],accel_mss,speed_ms,0,blend_radius_m)
    |   movel([0.157513, -1.375248, -2.579559, -0.757582, 1.570796, 1.728309],accel_mss,speed_ms,0,blend_radius_m)
    |   movel([0.157193, -1.374040, -2.580400, -0.757950, 1.570796, 1.727989],accel_mss,speed_ms,0,blend_radius_m)
    |   movel([0.156457, -1.372977, -2.581138, -0.758275, 1.570796, 1.727253],accel_mss,speed_ms,0,blend_radius_m)
    |   movel([0.155420, -1.372064, -2.581770, -0.758555, 1.570796, 1.726216],accel_mss,speed_ms,0,blend_radius_m)
    |   movel([0.154186, -1.371301, -2.582298, -0.758790, 1.570796, 1.724983],accel_mss,speed_ms,0,blend_radius_m)
    |   movel([0.152871, -1.370692, -2.582719, -0.758978, 1.570796, 1.723667],accel_mss,speed_ms,0,blend_radius_m)
    |   movel([0.150431, -1.369939, -2.583238, -0.759212, 1.570796, 1.721227],accel_mss,speed_ms,0,blend_radius_m)
    |   movel([0.151711, -1.372333, -2.581584, -0.758472, 1.570796, 1.722507],accel_mss,speed_ms,0,blend_radius_m)
    |   movel([0.152093, -1.373709, -2.580630, -0.758051, 1.570796, 1.722889],accel_mss,speed_ms,0,blend_radius_m)
    |   movel([0.152082, -1.375138, -2.579636, -0.757616, 1.570796, 1.722878],accel_mss,speed_ms,0,blend_radius_m)
    |   movel([0.151076, -1.375143, -2.579632, -0.757614, 1.570796, 1.721873],accel_mss,speed_ms,0,blend_radius_m)
    |   movel([0.150127, -1.374986, -2.579741, -0.757662, 1.570796, 1.720924],accel_mss,speed_ms,0,blend_radius_m)
    |   movel([0.148305, -1.374399, -2.580150, -0.757840, 1.570796, 1.719102],accel_mss,speed_ms,0,blend_radius_m)
    |   movel([0.146442, -1.373792, -2.580572, -0.758025, 1.570796, 1.717238],accel_mss,speed_ms,0,blend_radius_m)
    |   movel([0.145440, -1.373612, -2.580697, -0.758080, 1.570796, 1.716237],accel_mss,speed_ms,0,blend_radius_m)
    |   movel([0.144367, -1.373580, -2.580719, -0.758090, 1.570796, 1.715164],accel_mss,speed_ms,0,blend_radius_m)
    |   movel([0.143551, -1.375225, -2.579574, -0.757589, 1.570796, 1.714347],accel_mss,speed_ms,0,blend_radius_m)
    |   movel([0.143109, -1.376847, -2.578443, -0.757099, 1.570796, 1.713906],accel_mss,speed_ms,0,blend_radius_m)
    |   movel([0.141632, -1.376981, -2.578349, -0.757059, 1.570796, 1.712428],accel_mss,speed_ms,0,blend_radius_m)
    |   movel([0.140249, -1.376898, -2.578407, -0.757084, 1.570796, 1.711046],accel_mss,speed_ms,0,blend_radius_m)
    |   movel([0.138990, -1.376599, -2.578616, -0.757174, 1.570796, 1.709786],accel_mss,speed_ms,0,blend_radius_m)
    |   movel([0.137889, -1.376092, -2.578970, -0.757327, 1.570796, 1.708686],accel_mss,speed_ms,0,blend_radius_m)
    |   movel([0.137736, -1.376253, -2.578858, -0.757278, 1.570796, 1.708532],accel_mss,speed_ms,0,blend_radius_m)
    |   movel([0.136582, -1.378300, -2.577426, -0.756664, 1.570796, 1.707378],accel_mss,speed_ms,0,blend_radius_m)
    |   movel([0.135285, -1.380861, -2.575625, -0.755903, 1.570796, 1.706081],accel_mss,speed_ms,0,blend_radius_m)
    |   movel([0.134845, -1.382100, -2.574750, -0.755538, 1.570796, 1.705641],accel_mss,speed_ms,0,blend_radius_m)
    |   movel([0.134563, -1.383239, -2.573945, -0.755205, 1.570796, 1.705360],accel_mss,speed_ms,0,blend_radius_m)
    |   movel([0.134289, -1.385555, -2.572300, -0.754534, 1.570796, 1.705086],accel_mss,speed_ms,0,blend_radius_m)
    |   movel([0.130528, -1.383267, -2.573924, -0.755197, 1.570796, 1.701324],accel_mss,speed_ms,0,blend_radius_m)
    |   movel([0.129999, -1.384572, -2.572999, -0.754818, 1.570796, 1.700795],accel_mss,speed_ms,0,blend_radius_m)
    |   movel([0.129595, -1.385877, -2.572071, -0.754441, 1.570796, 1.700392],accel_mss,speed_ms,0,blend_radius_m)
    |   movel([0.129117, -1.388463, -2.570224, -0.753701, 1.570796, 1.699913],accel_mss,speed_ms,0,blend_radius_m)
    |   movel([0.129025, -1.390942, -2.568445, -0.753002, 1.570796, 1.699821],accel_mss,speed_ms,0,blend_radius_m)
    |   movel([0.129303, -1.393940, -2.566281, -0.752167, 1.570796, 1.700099],accel_mss,speed_ms,0,blend_radius_m)
    |   movel([0.129228, -1.394310, -2.566014, -0.752065, 1.570796, 1.700025],accel_mss,speed_ms,0,blend_radius_m)
    |   movel([0.129033, -1.394681, -2.565745, -0.751963, 1.570796, 1.699830],accel_mss,speed_ms,0,blend_radius_m)
    |   movel([0.128582, -1.395118, -2.565428, -0.751843, 1.570796, 1.699378],accel_mss,speed_ms,0,blend_radius_m)
    |   movel([0.124997, -1.397300, -2.563841, -0.751248, 1.570796, 1.695793],accel_mss,speed_ms,0,blend_radius_m)
    |   movel([0.123122, -1.398184, -2.563196, -0.751009, 1.570796, 1.693918],accel_mss,speed_ms,0,blend_radius_m)
    |   movel([0.122408, -1.398365, -2.563064, -0.750960, 1.570796, 1.693204],accel_mss,speed_ms,0,blend_radius_m)
    |   movel([0.121962, -1.398274, -2.563130, -0.750984, 1.570796, 1.692758],accel_mss,speed_ms,0,blend_radius_m)
    |   movel([0.123857, -1.399633, -2.562137, -0.750619, 1.570796, 1.694654],accel_mss,speed_ms,0,blend_radius_m)
    |   movel([0.124933, -1.400176, -2.561739, -0.750474, 1.570796, 1.695729],accel_mss,speed_ms,0,blend_radius_m)
    |   movel([0.126084, -1.400628, -2.561407, -0.750353, 1.570796, 1.696880],accel_mss,speed_ms,0,blend_radius_m)
    |   movel([0.123169, -1.403458, -2.559325, -0.749606, 1.570796, 1.693965],accel_mss,speed_ms,0,blend_radius_m)
    |   movel([0.120114, -1.406637, -2.556972, -0.748780, 1.570796, 1.690911],accel_mss,speed_ms,0,blend_radius_m)
    |   movel([0.118691, -1.408283, -2.555747, -0.748358, 1.570796, 1.689488],accel_mss,speed_ms,0,blend_radius_m)
    |   movel([0.117418, -1.409923, -2.554523, -0.747942, 1.570796, 1.688215],accel_mss,speed_ms,0,blend_radius_m)
    |   movel([0.116359, -1.411531, -2.553320, -0.747538, 1.570796, 1.687155],accel_mss,speed_ms,0,blend_radius_m)
    |   movel([0.115572, -1.413073, -2.552162, -0.747154, 1.570796, 1.686369],accel_mss,speed_ms,0,blend_radius_m)
    |   movel([0.117027, -1.412087, -2.552902, -0.747399, 1.570796, 1.687824],accel_mss,speed_ms,0,blend_radius_m)
    |   movel([0.118535, -1.411228, -2.553547, -0.747614, 1.570796, 1.689331],accel_mss,speed_ms,0,blend_radius_m)
    |   movel([0.120080, -1.410517, -2.554080, -0.747793, 1.570796, 1.690877],accel_mss,speed_ms,0,blend_radius_m)
    |   movel([0.121657, -1.409975, -2.554485, -0.747929, 1.570796, 1.692454],accel_mss,speed_ms,0,blend_radius_m)
    |   movel([0.120676, -1.410812, -2.553859, -0.747718, 1.570796, 1.691472],accel_mss,speed_ms,0,blend_radius_m)
    |   movel([0.118926, -1.412636, -2.552491, -0.747263, 1.570796, 1.689722],accel_mss,speed_ms,0,blend_radius_m)
    |   movel([0.118168, -1.413607, -2.551760, -0.747022, 1.570796, 1.688964],accel_mss,speed_ms,0,blend_radius_m)
    |   movel([0.116922, -1.415610, -2.550249, -0.746530, 1.570796, 1.687718],accel_mss,speed_ms,0,blend_radius_m)
    |   movel([0.116445, -1.416628, -2.549479, -0.746283, 1.570796, 1.687241],accel_mss,speed_ms,0,blend_radius_m)
    |   movel([0.116076, -1.417641, -2.548711, -0.746038, 1.570796, 1.686872],accel_mss,speed_ms,0,blend_radius_m)
    |   speed_ms = 0.005
    |   movel([0.116076, -1.409132, -2.544879, -0.758378, 1.570796, 1.686872],accel_mss,speed_ms,0,blend_radius_m)
    |   speed_ms = 0.040
    |   movel([0.122156, -1.411206, -2.543322, -0.757860, 1.570796, 1.692952],accel_mss,speed_ms,0,blend_radius_m)
    |   speed_ms = 0.005
    |   movel([0.122156, -1.419699, -2.547145, -0.745545, 1.570796, 1.692952],accel_mss,speed_ms,0,blend_radius_m)
    |   speed_ms = 0.025
    |   movel([0.122317, -1.418354, -2.548169, -0.745866, 1.570796, 1.693114],accel_mss,speed_ms,0,blend_radius_m)
    |   movel([0.122615, -1.416965, -2.549223, -0.746201, 1.570796, 1.693411],accel_mss,speed_ms,0,blend_radius_m)
    |   movel([0.123047, -1.415546, -2.550297, -0.746546, 1.570796, 1.693843],accel_mss,speed_ms,0,blend_radius_m)
    |   movel([0.123612, -1.414114, -2.551378, -0.746897, 1.570796, 1.694408],accel_mss,speed_ms,0,blend_radius_m)
    |   movel([0.124311, -1.412680, -2.552457, -0.747252, 1.570796, 1.695107],accel_mss,speed_ms,0,blend_radius_m)
    |   movel([0.125140, -1.411260, -2.553523, -0.747606, 1.570796, 1.695936],accel_mss,speed_ms,0,blend_radius_m)
    |   movel([0.126098, -1.409867, -2.554565, -0.747956, 1.570796, 1.696894],accel_mss,speed_ms,0,blend_radius_m)
    |   movel([0.127185, -1.408517, -2.555573, -0.748299, 1.570796, 1.697981],accel_mss,speed_ms,0,blend_radius_m)
    |   movel([0.130795, -1.404407, -2.558624, -0.749358, 1.570796, 1.701591],accel_mss,speed_ms,0,blend_radius_m)
    |   movel([0.131508, -1.403416, -2.559356, -0.749617, 1.570796, 1.702304],accel_mss,speed_ms,0,blend_radius_m)
    |   movel([0.132119, -1.402373, -2.560125, -0.749891, 1.570796, 1.702916],accel_mss,speed_ms,0,blend_radius_m)
    |   movel([0.132618, -1.401247, -2.560953, -0.750189, 1.570796, 1.703414],accel_mss,speed_ms,0,blend_radius_m)
    |   movel([0.132992, -1.400003, -2.561866, -0.750520, 1.570796, 1.703789],accel_mss,speed_ms,0,blend_radius_m)
    |   movel([0.133622, -1.396463, -2.564450, -0.751475, 1.570796, 1.704418],accel_mss,speed_ms,0,blend_radius_m)
    |   movel([0.134034, -1.394683, -2.565744, -0.751963, 1.570796, 1.704830],accel_mss,speed_ms,0,blend_radius_m)
    |   movel([0.134738, -1.392871, -2.567055, -0.752463, 1.570796, 1.705535],accel_mss,speed_ms,0,blend_radius_m)
    |   movel([0.135359, -1.391780, -2.567842, -0.752767, 1.570796, 1.706155],accel_mss,speed_ms,0,blend_radius_m)
    |   movel([0.136104, -1.390718, -2.568607, -0.753064, 1.570796, 1.706901],accel_mss,speed_ms,0,blend_radius_m)
    |   movel([0.137895, -1.388684, -2.570066, -0.753639, 1.570796, 1.708691],accel_mss,speed_ms,0,blend_radius_m)
    |   movel([0.139949, -1.386753, -2.571446, -0.754189, 1.570796, 1.710746],accel_mss,speed_ms,0,blend_radius_m)
    |   movel([0.142116, -1.384910, -2.572759, -0.754720, 1.570796, 1.712913],accel_mss,speed_ms,0,blend_radius_m)
    |   movel([0.144257, -1.383180, -2.573986, -0.755222, 1.570796, 1.715054],accel_mss,speed_ms,0,blend_radius_m)
    |   movel([0.146504, -1.381588, -2.575112, -0.755689, 1.570796, 1.717300],accel_mss,speed_ms,0,blend_radius_m)
    |   movel([0.147652, -1.380911, -2.575590, -0.755888, 1.570796, 1.718449],accel_mss,speed_ms,0,blend_radius_m)
    |   movel([0.148814, -1.380344, -2.575989, -0.756056, 1.570796, 1.719611],accel_mss,speed_ms,0,blend_radius_m)
    |   movel([0.149977, -1.379920, -2.576288, -0.756181, 1.570796, 1.720774],accel_mss,speed_ms,0,blend_radius_m)
    |   movel([0.151144, -1.379659, -2.576471, -0.756259, 1.570796, 1.721940],accel_mss,speed_ms,0,blend_radius_m)
    |   speed_ms = 0.005
    |   movel([0.151144, -1.370871, -2.572475, -0.769043, 1.570796, 1.721940],accel_mss,speed_ms,0,blend_radius_m)
    |   speed_ms = 0.040
    |   movel([0.152596, -1.371799, -2.571830, -0.768760, 1.570796, 1.723392],accel_mss,speed_ms,0,blend_radius_m)
    |   speed_ms = 0.005
    |   movel([0.152596, -1.380580, -2.575823, -0.755986, 1.570796, 1.723392],accel_mss,speed_ms,0,blend_radius_m)
    |   speed_ms = 0.025
    |   movel([0.153054, -1.380821, -2.575653, -0.755915, 1.570796, 1.723850],accel_mss,speed_ms,0,blend_radius_m)
    |   movel([0.153672, -1.381254, -2.575348, -0.755787, 1.570796, 1.724468],accel_mss,speed_ms,0,blend_radius_m)
    |   movel([0.154640, -1.382595, -2.574401, -0.755394, 1.570796, 1.725436],accel_mss,speed_ms,0,blend_radius_m)
    |   movel([0.154958, -1.383386, -2.573840, -0.755162, 1.570796, 1.725754],accel_mss,speed_ms,0,blend_radius_m)
    |   movel([0.154970, -1.383817, -2.573535, -0.755037, 1.570796, 1.725766],accel_mss,speed_ms,0,blend_radius_m)
    |   movel([0.154856, -1.383924, -2.573459, -0.755006, 1.570796, 1.725652],accel_mss,speed_ms,0,blend_radius_m)
    |   movel([0.154626, -1.383914, -2.573466, -0.755009, 1.570796, 1.725423],accel_mss,speed_ms,0,blend_radius_m)
    |   movel([0.152311, -1.383179, -2.573987, -0.755223, 1.570796, 1.723107],accel_mss,speed_ms,0,blend_radius_m)
    |   movel([0.151023, -1.383010, -2.574107, -0.755272, 1.570796, 1.721819],accel_mss,speed_ms,0,blend_radius_m)
    |   movel([0.150328, -1.383065, -2.574068, -0.755256, 1.570796, 1.721124],accel_mss,speed_ms,0,blend_radius_m)
    |   movel([0.149590, -1.383242, -2.573942, -0.755204, 1.570796, 1.720387],accel_mss,speed_ms,0,blend_radius_m)
    |   movel([0.148758, -1.383600, -2.573689, -0.755100, 1.570796, 1.719554],accel_mss,speed_ms,0,blend_radius_m)
    |   movel([0.147944, -1.384063, -2.573360, -0.754965, 1.570796, 1.718741],accel_mss,speed_ms,0,blend_radius_m)
    |   movel([0.146001, -1.385362, -2.572438, -0.754589, 1.570796, 1.716797],accel_mss,speed_ms,0,blend_radius_m)
    |   movel([0.144120, -1.386826, -2.571395, -0.754169, 1.570796, 1.714917],accel_mss,speed_ms,0,blend_radius_m)
    |   movel([0.142359, -1.388408, -2.570264, -0.753717, 1.570796, 1.713155],accel_mss,speed_ms,0,blend_radius_m)
    |   movel([0.140776, -1.390055, -2.569083, -0.753251, 1.570796, 1.711573],accel_mss,speed_ms,0,blend_radius_m)
    |   movel([0.142033, -1.391913, -2.567746, -0.752730, 1.570796, 1.712830],accel_mss,speed_ms,0,blend_radius_m)
    |   movel([0.142978, -1.393974, -2.566257, -0.752158, 1.570796, 1.713775],accel_mss,speed_ms,0,blend_radius_m)
    |   movel([0.142113, -1.393657, -2.566487, -0.752246, 1.570796, 1.712909],accel_mss,speed_ms,0,blend_radius_m)
    |   movel([0.141125, -1.393522, -2.566584, -0.752283, 1.570796, 1.711921],accel_mss,speed_ms,0,blend_radius_m)
    |   movel([0.140044, -1.393579, -2.566543, -0.752267, 1.570796, 1.710840],accel_mss,speed_ms,0,blend_radius_m)
    |   movel([0.138909, -1.393824, -2.566366, -0.752199, 1.570796, 1.709705],accel_mss,speed_ms,0,blend_radius_m)
    |   movel([0.138385, -1.394098, -2.566167, -0.752124, 1.570796, 1.709181],accel_mss,speed_ms,0,blend_radius_m)
    |   movel([0.138191, -1.394517, -2.565864, -0.752008, 1.570796, 1.708987],accel_mss,speed_ms,0,blend_radius_m)
    |   movel([0.137202, -1.399012, -2.562591, -0.750786, 1.570796, 1.707998],accel_mss,speed_ms,0,blend_radius_m)
    |   movel([0.136495, -1.401317, -2.560901, -0.750170, 1.570796, 1.707291],accel_mss,speed_ms,0,blend_radius_m)
    |   movel([0.135588, -1.403671, -2.559168, -0.749550, 1.570796, 1.706385],accel_mss,speed_ms,0,blend_radius_m)
    |   movel([0.134479, -1.406011, -2.557437, -0.748942, 1.570796, 1.705276],accel_mss,speed_ms,0,blend_radius_m)
    |   movel([0.133160, -1.408278, -2.555751, -0.748360, 1.570796, 1.703956],accel_mss,speed_ms,0,blend_radius_m)
    |   movel([0.130327, -1.412803, -2.552365, -0.747221, 1.570796, 1.701124],accel_mss,speed_ms,0,blend_radius_m)
    |   movel([0.129193, -1.415062, -2.550663, -0.746664, 1.570796, 1.699989],accel_mss,speed_ms,0,blend_radius_m)
    |   movel([0.128418, -1.417347, -2.548934, -0.746109, 1.570796, 1.699215],accel_mss,speed_ms,0,blend_radius_m)
    |   speed_ms = 0.005
    |   movel([0.128418, -1.408836, -2.545101, -0.758452, 1.570796, 1.699215],accel_mss,speed_ms,0,blend_radius_m)
    |   speed_ms = 0.040
    |   movel([0.140039, -1.404533, -2.548309, -0.759547, 1.570796, 1.710835],accel_mss,speed_ms,0,blend_radius_m)
    |   speed_ms = 0.005
    |   movel([0.140039, -1.413076, -2.552160, -0.747153, 1.570796, 1.710835],accel_mss,speed_ms,0,blend_radius_m)
    |   speed_ms = 0.025
    |   movel([0.139433, -1.414923, -2.550768, -0.746698, 1.570796, 1.710229],accel_mss,speed_ms,0,blend_radius_m)
    |   movel([0.138485, -1.416772, -2.549370, -0.746248, 1.570796, 1.709281],accel_mss,speed_ms,0,blend_radius_m)
    |   movel([0.137230, -1.418562, -2.548011, -0.745816, 1.570796, 1.708026],accel_mss,speed_ms,0,blend_radius_m)
    |   movel([0.135707, -1.420236, -2.546736, -0.745417, 1.570796, 1.706503],accel_mss,speed_ms,0,blend_radius_m)
    |   speed_ms = 0.005
    |   movel([0.135707, -1.411747, -2.542915, -0.757727, 1.570796, 1.706503],accel_mss,speed_ms,0,blend_radius_m)
    |   speed_ms = 0.040
    |   movel([0.133094, -1.409626, -2.544509, -0.758254, 1.570796, 1.703890],accel_mss,speed_ms,0,blend_radius_m)
    |   speed_ms = 0.005
    |   movel([0.133094, -1.418131, -2.548338, -0.745920, 1.570796, 1.703890],accel_mss,speed_ms,0,blend_radius_m)
    |   speed_ms = 0.025
    |   movel([0.125803, -1.429512, -2.539594, -0.743283, 1.570796, 1.696599],accel_mss,speed_ms,0,blend_radius_m)
    |   movel([0.125462, -1.430249, -2.539022, -0.743119, 1.570796, 1.696259],accel_mss,speed_ms,0,blend_radius_m)
    |   movel([0.125623, -1.431031, -2.538412, -0.742945, 1.570796, 1.696420],accel_mss,speed_ms,0,blend_radius_m)
    |   movel([0.125828, -1.432042, -2.537624, -0.742723, 1.570796, 1.696624],accel_mss,speed_ms,0,blend_radius_m)
    |   movel([0.125738, -1.433161, -2.536749, -0.742479, 1.570796, 1.696535],accel_mss,speed_ms,0,blend_radius_m)
    |   speed_ms = 0.005
    |   movel([0.125738, -1.424771, -2.532984, -0.754634, 1.570796, 1.696535],accel_mss,speed_ms,0,blend_radius_m)
    |   speed_ms = 0.040
    |   movel([0.138899, -1.417950, -2.538217, -0.756222, 1.570796, 1.709695],accel_mss,speed_ms,0,blend_radius_m)
    |   speed_ms = 0.005
    |   movel([0.138899, -1.426392, -2.542011, -0.743986, 1.570796, 1.709695],accel_mss,speed_ms,0,blend_radius_m)
    |   speed_ms = 0.025
    |   movel([0.139025, -1.425197, -2.542932, -0.744259, 1.570796, 1.709821],accel_mss,speed_ms,0,blend_radius_m)
    |   movel([0.139330, -1.423962, -2.543883, -0.744544, 1.570796, 1.710126],accel_mss,speed_ms,0,blend_radius_m)
    |   movel([0.139805, -1.422708, -2.544845, -0.744836, 1.570796, 1.710601],accel_mss,speed_ms,0,blend_radius_m)
    |   movel([0.140448, -1.421451, -2.545808, -0.745130, 1.570796, 1.711245],accel_mss,speed_ms,0,blend_radius_m)
    |   movel([0.140996, -1.420593, -2.546463, -0.745333, 1.570796, 1.711792],accel_mss,speed_ms,0,blend_radius_m)
    |   movel([0.141644, -1.419761, -2.547098, -0.745530, 1.570796, 1.712440],accel_mss,speed_ms,0,blend_radius_m)
    |   movel([0.142394, -1.418997, -2.547680, -0.745712, 1.570796, 1.713190],accel_mss,speed_ms,0,blend_radius_m)
    |   movel([0.143257, -1.418333, -2.548184, -0.745871, 1.570796, 1.714053],accel_mss,speed_ms,0,blend_radius_m)
    |   movel([0.144050, -1.417918, -2.548500, -0.745971, 1.570796, 1.714846],accel_mss,speed_ms,0,blend_radius_m)
    |   movel([0.144926, -1.417630, -2.548719, -0.746040, 1.570796, 1.715722],accel_mss,speed_ms,0,blend_radius_m)
    |   movel([0.145853, -1.417449, -2.548856, -0.746084, 1.570796, 1.716649],accel_mss,speed_ms,0,blend_radius_m)
    |   movel([0.146806, -1.417355, -2.548927, -0.746107, 1.570796, 1.717603],accel_mss,speed_ms,0,blend_radius_m)
    |   movel([0.148672, -1.417342, -2.548937, -0.746110, 1.570796, 1.719469],accel_mss,speed_ms,0,blend_radius_m)
    |   movel([0.150298, -1.417427, -2.548873, -0.746089, 1.570796, 1.721094],accel_mss,speed_ms,0,blend_radius_m)
    |   movel([0.149162, -1.417458, -2.548849, -0.746082, 1.570796, 1.719959],accel_mss,speed_ms,0,blend_radius_m)
    |   movel([0.147991, -1.417684, -2.548678, -0.746027, 1.570796, 1.718788],accel_mss,speed_ms,0,blend_radius_m)
    |   movel([0.146809, -1.418127, -2.548342, -0.745921, 1.570796, 1.717605],accel_mss,speed_ms,0,blend_radius_m)
    |   movel([0.145637, -1.418809, -2.547823, -0.745757, 1.570796, 1.716434],accel_mss,speed_ms,0,blend_radius_m)
    |   movel([0.144714, -1.419569, -2.547244, -0.745576, 1.570796, 1.715510],accel_mss,speed_ms,0,blend_radius_m)
    |   movel([0.143902, -1.420422, -2.546594, -0.745373, 1.570796, 1.714698],accel_mss,speed_ms,0,blend_radius_m)
    |   movel([0.143220, -1.421284, -2.545935, -0.745170, 1.570796, 1.714017],accel_mss,speed_ms,0,blend_radius_m)
    |   movel([0.142647, -1.422174, -2.545254, -0.744961, 1.570796, 1.713444],accel_mss,speed_ms,0,blend_radius_m)
    |   movel([0.141804, -1.424002, -2.543852, -0.744535, 1.570796, 1.712601],accel_mss,speed_ms,0,blend_radius_m)
    |   movel([0.141335, -1.425823, -2.542450, -0.744116, 1.570796, 1.712131],accel_mss,speed_ms,0,blend_radius_m)
    |   movel([0.141202, -1.427706, -2.540995, -0.743688, 1.570796, 1.711998],accel_mss,speed_ms,0,blend_radius_m)
    |   speed_ms = 0.005
    |   movel([0.141202, -1.419274, -2.537207, -0.755909, 1.570796, 1.711998],accel_mss,speed_ms,0,blend_radius_m)
    |   speed_ms = 0.040
    |   movel([0.144452, -1.414997, -2.540460, -0.756931, 1.570796, 1.715248],accel_mss,speed_ms,0,blend_radius_m)
    |   speed_ms = 0.005
    |   movel([0.144452, -1.423462, -2.544267, -0.744660, 1.570796, 1.715248],accel_mss,speed_ms,0,blend_radius_m)
    |   speed_ms = 0.025
    |   movel([0.144280, -1.423741, -2.544053, -0.744595, 1.570796, 1.715076],accel_mss,speed_ms,0,blend_radius_m)
    |   movel([0.143943, -1.423872, -2.543952, -0.744565, 1.570796, 1.714739],accel_mss,speed_ms,0,blend_radius_m)
    |   movel([0.143725, -1.423742, -2.544052, -0.744595, 1.570796, 1.714521],accel_mss,speed_ms,0,blend_radius_m)
    |   movel([0.143688, -1.423468, -2.544262, -0.744659, 1.570796, 1.714484],accel_mss,speed_ms,0,blend_radius_m)
    |   movel([0.144043, -1.422862, -2.544728, -0.744800, 1.570796, 1.714839],accel_mss,speed_ms,0,blend_radius_m)
    |   movel([0.144301, -1.422629, -2.544906, -0.744854, 1.570796, 1.715097],accel_mss,speed_ms,0,blend_radius_m)
    |   movel([0.144609, -1.422592, -2.544934, -0.744863, 1.570796, 1.715405],accel_mss,speed_ms,0,blend_radius_m)
    |   movel([0.144782, -1.422774, -2.544795, -0.744820, 1.570796, 1.715578],accel_mss,speed_ms,0,blend_radius_m)
    |   movel([0.144654, -1.423361, -2.544344, -0.744684, 1.570796, 1.715450],accel_mss,speed_ms,0,blend_radius_m)
    |   speed_ms = 0.005
    |   movel([0.144654, -1.414896, -2.540537, -0.756956, 1.570796, 1.715450],accel_mss,speed_ms,0,blend_radius_m)
    |   speed_ms = 0.040
    |   movel([0.144507, -1.422432, -2.534786, -0.755171, 1.570796, 1.715303],accel_mss,speed_ms,0,blend_radius_m)
    |   speed_ms = 0.005
    |   movel([0.144507, -1.430840, -2.538561, -0.742988, 1.570796, 1.715303],accel_mss,speed_ms,0,blend_radius_m)
    |   speed_ms = 0.025
    |   movel([0.145589, -1.429791, -2.539377, -0.743220, 1.570796, 1.716386],accel_mss,speed_ms,0,blend_radius_m)
    |   movel([0.146479, -1.428689, -2.540233, -0.743467, 1.570796, 1.717275],accel_mss,speed_ms,0,blend_radius_m)
    |   movel([0.148259, -1.426466, -2.541954, -0.743969, 1.570796, 1.719056],accel_mss,speed_ms,0,blend_radius_m)
    |   movel([0.149797, -1.425018, -2.543070, -0.744301, 1.570796, 1.720593],accel_mss,speed_ms,0,blend_radius_m)
    |   movel([0.154970, -1.420887, -2.546238, -0.745263, 1.570796, 1.725767],accel_mss,speed_ms,0,blend_radius_m)
    |   movel([0.155933, -1.419940, -2.546961, -0.745487, 1.570796, 1.726729],accel_mss,speed_ms,0,blend_radius_m)
    |   movel([0.156229, -1.419442, -2.547341, -0.745606, 1.570796, 1.727025],accel_mss,speed_ms,0,blend_radius_m)
    |   movel([0.156268, -1.418979, -2.547693, -0.745716, 1.570796, 1.727065],accel_mss,speed_ms,0,blend_radius_m)
    |   movel([0.155923, -1.418597, -2.547984, -0.745808, 1.570796, 1.726719],accel_mss,speed_ms,0,blend_radius_m)
    |   movel([0.155351, -1.418416, -2.548122, -0.745851, 1.570796, 1.726147],accel_mss,speed_ms,0,blend_radius_m)
    |   movel([0.154425, -1.418285, -2.548221, -0.745883, 1.570796, 1.725222],accel_mss,speed_ms,0,blend_radius_m)
    |   movel([0.153507, -1.418347, -2.548174, -0.745868, 1.570796, 1.724303],accel_mss,speed_ms,0,blend_radius_m)
    |   movel([0.152532, -1.418622, -2.547965, -0.745802, 1.570796, 1.723329],accel_mss,speed_ms,0,blend_radius_m)
    |   movel([0.151442, -1.419129, -2.547579, -0.745681, 1.570796, 1.722238],accel_mss,speed_ms,0,blend_radius_m)
    |   movel([0.150307, -1.419846, -2.547033, -0.745510, 1.570796, 1.721103],accel_mss,speed_ms,0,blend_radius_m)
    |   movel([0.149219, -1.420725, -2.546362, -0.745301, 1.570796, 1.720015],accel_mss,speed_ms,0,blend_radius_m)
    |   movel([0.148183, -1.421722, -2.545600, -0.745067, 1.570796, 1.718979],accel_mss,speed_ms,0,blend_radius_m)
    |   movel([0.147203, -1.422803, -2.544772, -0.744814, 1.570796, 1.718000],accel_mss,speed_ms,0,blend_radius_m)
    |   movel([0.145436, -1.425046, -2.543049, -0.744294, 1.570796, 1.716233],accel_mss,speed_ms,0,blend_radius_m)
    |   movel([0.143956, -1.427141, -2.541432, -0.743816, 1.570796, 1.714753],accel_mss,speed_ms,0,blend_radius_m)
    |   movel([0.141364, -1.431051, -2.538397, -0.742941, 1.570796, 1.712160],accel_mss,speed_ms,0,blend_radius_m)
    |   movel([0.140408, -1.432317, -2.537409, -0.742663, 1.570796, 1.711204],accel_mss,speed_ms,0,blend_radius_m)
    |   movel([0.139318, -1.433538, -2.536454, -0.742397, 1.570796, 1.710114],accel_mss,speed_ms,0,blend_radius_m)
    |   movel([0.138085, -1.434659, -2.535576, -0.742154, 1.570796, 1.708881],accel_mss,speed_ms,0,blend_radius_m)
    |   movel([0.136732, -1.435606, -2.534831, -0.741951, 1.570796, 1.707529],accel_mss,speed_ms,0,blend_radius_m)
    |   movel([0.135286, -1.436308, -2.534279, -0.741801, 1.570796, 1.706082],accel_mss,speed_ms,0,blend_radius_m)
    |   movel([0.136405, -1.436160, -2.534396, -0.741833, 1.570796, 1.707202],accel_mss,speed_ms,0,blend_radius_m)
    |   movel([0.137549, -1.435904, -2.534597, -0.741888, 1.570796, 1.708345],accel_mss,speed_ms,0,blend_radius_m)
    |   movel([0.138706, -1.435541, -2.534883, -0.741965, 1.570796, 1.709502],accel_mss,speed_ms,0,blend_radius_m)
    |   movel([0.139857, -1.435078, -2.535247, -0.742064, 1.570796, 1.710653],accel_mss,speed_ms,0,blend_radius_m)
    |   movel([0.139795, -1.436195, -2.534368, -0.741825, 1.570796, 1.710591],accel_mss,speed_ms,0,blend_radius_m)
    |   movel([0.139527, -1.437360, -2.533450, -0.741578, 1.570796, 1.710323],accel_mss,speed_ms,0,blend_radius_m)
    |   movel([0.139063, -1.438543, -2.532516, -0.741330, 1.570796, 1.709859],accel_mss,speed_ms,0,blend_radius_m)
    |   movel([0.138413, -1.439717, -2.531587, -0.741085, 1.570796, 1.709209],accel_mss,speed_ms,0,blend_radius_m)
    |   movel([0.139661, -1.438596, -2.532474, -0.741318, 1.570796, 1.710458],accel_mss,speed_ms,0,blend_radius_m)
    |   movel([0.140754, -1.437394, -2.533424, -0.741571, 1.570796, 1.711551],accel_mss,speed_ms,0,blend_radius_m)
    |   movel([0.141703, -1.436124, -2.534425, -0.741841, 1.570796, 1.712500],accel_mss,speed_ms,0,blend_radius_m)
    |   movel([0.142525, -1.434801, -2.535464, -0.742124, 1.570796, 1.713322],accel_mss,speed_ms,0,blend_radius_m)
    |   movel([0.142532, -1.435541, -2.534883, -0.741965, 1.570796, 1.713328],accel_mss,speed_ms,0,blend_radius_m)
    |   movel([0.142343, -1.436397, -2.534209, -0.741782, 1.570796, 1.713139],accel_mss,speed_ms,0,blend_radius_m)
    |   movel([0.140789, -1.440311, -2.531116, -0.740962, 1.570796, 1.711585],accel_mss,speed_ms,0,blend_radius_m)
    |   movel([0.140495, -1.441256, -2.530365, -0.740767, 1.570796, 1.711292],accel_mss,speed_ms,0,blend_radius_m)
    |   movel([0.140359, -1.442121, -2.529677, -0.740590, 1.570796, 1.711155],accel_mss,speed_ms,0,blend_radius_m)
    |   movel([0.141079, -1.440772, -2.530750, -0.740867, 1.570796, 1.711875],accel_mss,speed_ms,0,blend_radius_m)
    |   movel([0.141889, -1.439529, -2.531736, -0.741124, 1.570796, 1.712685],accel_mss,speed_ms,0,blend_radius_m)
    |   movel([0.143702, -1.437250, -2.533538, -0.741602, 1.570796, 1.714498],accel_mss,speed_ms,0,blend_radius_m)
    |   movel([0.145649, -1.435035, -2.535280, -0.742074, 1.570796, 1.716445],accel_mss,speed_ms,0,blend_radius_m)
    |   movel([0.147589, -1.432633, -2.537162, -0.742594, 1.570796, 1.718385],accel_mss,speed_ms,0,blend_radius_m)
    |   movel([0.148589, -1.431086, -2.538370, -0.742933, 1.570796, 1.719385],accel_mss,speed_ms,0,blend_radius_m)
    |   movel([0.149256, -1.430246, -2.539024, -0.743119, 1.570796, 1.720052],accel_mss,speed_ms,0,blend_radius_m)
    |   movel([0.149589, -1.429953, -2.539251, -0.743184, 1.570796, 1.720386],accel_mss,speed_ms,0,blend_radius_m)
    |   movel([0.149911, -1.429797, -2.539373, -0.743219, 1.570796, 1.720707],accel_mss,speed_ms,0,blend_radius_m)
    |   movel([0.150198, -1.429798, -2.539372, -0.743219, 1.570796, 1.720995],accel_mss,speed_ms,0,blend_radius_m)
    |   movel([0.150440, -1.429930, -2.539270, -0.743190, 1.570796, 1.721237],accel_mss,speed_ms,0,blend_radius_m)
    |   movel([0.150781, -1.430456, -2.538861, -0.743073, 1.570796, 1.721577],accel_mss,speed_ms,0,blend_radius_m)
    |   movel([0.150900, -1.431133, -2.538333, -0.742923, 1.570796, 1.721696],accel_mss,speed_ms,0,blend_radius_m)
    |   movel([0.150766, -1.431721, -2.537875, -0.742794, 1.570796, 1.721562],accel_mss,speed_ms,0,blend_radius_m)
    |   movel([0.151809, -1.429724, -2.539429, -0.743235, 1.570796, 1.722606],accel_mss,speed_ms,0,blend_radius_m)
    |   movel([0.152614, -1.427712, -2.540990, -0.743687, 1.570796, 1.723410],accel_mss,speed_ms,0,blend_radius_m)
    |   movel([0.153173, -1.425716, -2.542532, -0.744140, 1.570796, 1.723970],accel_mss,speed_ms,0,blend_radius_m)
    |   movel([0.153474, -1.423762, -2.544036, -0.744591, 1.570796, 1.724270],accel_mss,speed_ms,0,blend_radius_m)
    |   speed_ms = 0.005
    |   movel([0.153474, -1.415300, -2.540231, -0.756858, 1.570796, 1.724270],accel_mss,speed_ms,0,blend_radius_m)
    |   speed_ms = 0.040
    |   movel([0.155727, -1.415895, -2.539779, -0.756714, 1.570796, 1.726523],accel_mss,speed_ms,0,blend_radius_m)
    |   speed_ms = 0.005
    |   movel([0.155727, -1.424353, -2.543582, -0.744454, 1.570796, 1.726523],accel_mss,speed_ms,0,blend_radius_m)
    |   speed_ms = 0.025
    |   movel([0.157059, -1.424585, -2.543404, -0.744400, 1.570796, 1.727855],accel_mss,speed_ms,0,blend_radius_m)
    |   movel([0.157561, -1.424872, -2.543183, -0.744334, 1.570796, 1.728358],accel_mss,speed_ms,0,blend_radius_m)
    |   movel([0.157840, -1.425338, -2.542824, -0.744227, 1.570796, 1.728636],accel_mss,speed_ms,0,blend_radius_m)
    |   movel([0.157852, -1.425859, -2.542422, -0.744108, 1.570796, 1.728648],accel_mss,speed_ms,0,blend_radius_m)
    |   movel([0.155752, -1.434986, -2.535319, -0.742084, 1.570796, 1.726549],accel_mss,speed_ms,0,blend_radius_m)
    |   movel([0.155558, -1.435640, -2.534805, -0.741944, 1.570796, 1.726354],accel_mss,speed_ms,0,blend_radius_m)
    |   movel([0.155250, -1.436295, -2.534290, -0.741804, 1.570796, 1.726046],accel_mss,speed_ms,0,blend_radius_m)
    |   movel([0.154796, -1.436859, -2.533845, -0.741684, 1.570796, 1.725592],accel_mss,speed_ms,0,blend_radius_m)
    |   movel([0.154177, -1.437236, -2.533548, -0.741604, 1.570796, 1.724973],accel_mss,speed_ms,0,blend_radius_m)
    |   movel([0.153571, -1.437326, -2.533477, -0.741586, 1.570796, 1.724367],accel_mss,speed_ms,0,blend_radius_m)
    |   movel([0.152435, -1.437193, -2.533582, -0.741614, 1.570796, 1.723231],accel_mss,speed_ms,0,blend_radius_m)
    |   movel([0.151832, -1.437307, -2.533492, -0.741590, 1.570796, 1.722628],accel_mss,speed_ms,0,blend_radius_m)
    |   movel([0.151142, -1.437770, -2.533127, -0.741492, 1.570796, 1.721939],accel_mss,speed_ms,0,blend_radius_m)
    |   movel([0.150541, -1.438373, -2.532651, -0.741365, 1.570796, 1.721338],accel_mss,speed_ms,0,blend_radius_m)
    |   movel([0.149774, -1.439036, -2.532126, -0.741227, 1.570796, 1.720570],accel_mss,speed_ms,0,blend_radius_m)
    |   movel([0.148924, -1.439586, -2.531691, -0.741112, 1.570796, 1.719720],accel_mss,speed_ms,0,blend_radius_m)
    |   movel([0.148026, -1.440014, -2.531351, -0.741023, 1.570796, 1.718822],accel_mss,speed_ms,0,blend_radius_m)
    |   movel([0.147111, -1.440313, -2.531115, -0.740961, 1.570796, 1.717907],accel_mss,speed_ms,0,blend_radius_m)
    |   movel([0.146210, -1.440474, -2.530987, -0.740928, 1.570796, 1.717007],accel_mss,speed_ms,0,blend_radius_m)
    |   movel([0.145362, -1.440487, -2.530976, -0.740925, 1.570796, 1.716158],accel_mss,speed_ms,0,blend_radius_m)
    |   movel([0.144595, -1.440349, -2.531086, -0.740954, 1.570796, 1.715391],accel_mss,speed_ms,0,blend_radius_m)
    |   movel([0.143942, -1.440045, -2.531327, -0.741017, 1.570796, 1.714738],accel_mss,speed_ms,0,blend_radius_m)
    |   speed_ms = 0.005
    |   movel([0.143942, -1.431708, -2.527591, -0.753090, 1.570796, 1.714738],accel_mss,speed_ms,0,blend_radius_m)
    |   speed_ms = 0.040
    |   movel([0.137204, -1.440206, -2.520886, -0.751298, 1.570796, 1.708000],accel_mss,speed_ms,0,blend_radius_m)
    |   speed_ms = 0.005
    |   movel([0.137204, -1.448477, -2.524587, -0.739325, 1.570796, 1.708000],accel_mss,speed_ms,0,blend_radius_m)
    |   speed_ms = 0.025
    |   movel([0.137019, -1.457046, -2.517625, -0.737718, 1.570796, 1.707815],accel_mss,speed_ms,0,blend_radius_m)
    |   movel([0.136871, -1.458122, -2.516743, -0.737524, 1.570796, 1.707667],accel_mss,speed_ms,0,blend_radius_m)
    |   movel([0.136626, -1.458650, -2.516310, -0.737430, 1.570796, 1.707422],accel_mss,speed_ms,0,blend_radius_m)
    |   movel([0.136206, -1.459122, -2.515921, -0.737346, 1.570796, 1.707002],accel_mss,speed_ms,0,blend_radius_m)
    |   movel([0.135025, -1.459935, -2.515252, -0.737202, 1.570796, 1.705822],accel_mss,speed_ms,0,blend_radius_m)
    |   movel([0.134683, -1.460492, -2.514793, -0.737104, 1.570796, 1.705479],accel_mss,speed_ms,0,blend_radius_m)
    |   movel([0.134582, -1.461067, -2.514319, -0.737003, 1.570796, 1.705378],accel_mss,speed_ms,0,blend_radius_m)
    |   movel([0.134732, -1.461934, -2.513603, -0.736852, 1.570796, 1.705529],accel_mss,speed_ms,0,blend_radius_m)
    |   movel([0.135154, -1.462700, -2.512969, -0.736720, 1.570796, 1.705950],accel_mss,speed_ms,0,blend_radius_m)
    |   movel([0.136182, -1.464074, -2.511830, -0.736484, 1.570796, 1.706978],accel_mss,speed_ms,0,blend_radius_m)
    |   movel([0.136635, -1.465118, -2.510963, -0.736308, 1.570796, 1.707432],accel_mss,speed_ms,0,blend_radius_m)
    |   movel([0.137017, -1.466723, -2.509627, -0.736040, 1.570796, 1.707813],accel_mss,speed_ms,0,blend_radius_m)
    |   movel([0.137025, -1.467498, -2.508980, -0.735911, 1.570796, 1.707822],accel_mss,speed_ms,0,blend_radius_m)
    |   movel([0.136828, -1.468134, -2.508448, -0.735807, 1.570796, 1.707624],accel_mss,speed_ms,0,blend_radius_m)
    |   movel([0.136632, -1.468368, -2.508253, -0.735769, 1.570796, 1.707428],accel_mss,speed_ms,0,blend_radius_m)
    |   movel([0.136362, -1.468533, -2.508115, -0.735742, 1.570796, 1.707158],accel_mss,speed_ms,0,blend_radius_m)
    |   movel([0.136010, -1.468616, -2.508045, -0.735728, 1.570796, 1.706806],accel_mss,speed_ms,0,blend_radius_m)
    |   movel([0.135569, -1.468605, -2.508054, -0.735730, 1.570796, 1.706365],accel_mss,speed_ms,0,blend_radius_m)
    |   movel([0.135443, -1.469284, -2.507485, -0.735620, 1.570796, 1.706240],accel_mss,speed_ms,0,blend_radius_m)
    |   movel([0.135517, -1.470011, -2.506875, -0.735502, 1.570796, 1.706313],accel_mss,speed_ms,0,blend_radius_m)
    |   movel([0.136079, -1.471508, -2.505618, -0.735263, 1.570796, 1.706875],accel_mss,speed_ms,0,blend_radius_m)
    |   movel([0.136903, -1.472886, -2.504456, -0.735047, 1.570796, 1.707699],accel_mss,speed_ms,0,blend_radius_m)
    |   movel([0.137648, -1.473937, -2.503569, -0.734883, 1.570796, 1.708444],accel_mss,speed_ms,0,blend_radius_m)
    |   movel([0.138676, -1.474965, -2.502699, -0.734725, 1.570796, 1.709472],accel_mss,speed_ms,0,blend_radius_m)
    |   movel([0.139889, -1.475927, -2.501883, -0.734579, 1.570796, 1.710685],accel_mss,speed_ms,0,blend_radius_m)
    |   movel([0.140905, -1.477006, -2.500967, -0.734416, 1.570796, 1.711701],accel_mss,speed_ms,0,blend_radius_m)
    |   movel([0.141221, -1.477642, -2.500426, -0.734321, 1.570796, 1.712017],accel_mss,speed_ms,0,blend_radius_m)
    |   movel([0.141345, -1.478374, -2.499803, -0.734212, 1.570796, 1.712141],accel_mss,speed_ms,0,blend_radius_m)
    |   movel([0.141282, -1.478790, -2.499447, -0.734151, 1.570796, 1.712078],accel_mss,speed_ms,0,blend_radius_m)
    |   movel([0.141089, -1.479219, -2.499082, -0.734088, 1.570796, 1.711886],accel_mss,speed_ms,0,blend_radius_m)
    |   movel([0.140781, -1.479565, -2.498787, -0.734038, 1.570796, 1.711578],accel_mss,speed_ms,0,blend_radius_m)
    |   movel([0.140371, -1.479740, -2.498637, -0.734012, 1.570796, 1.711168],accel_mss,speed_ms,0,blend_radius_m)
    |   movel([0.140056, -1.479702, -2.498669, -0.734018, 1.570796, 1.710852],accel_mss,speed_ms,0,blend_radius_m)
    |   movel([0.139804, -1.479567, -2.498784, -0.734037, 1.570796, 1.710600],accel_mss,speed_ms,0,blend_radius_m)
    |   movel([0.137707, -1.477964, -2.500152, -0.734273, 1.570796, 1.708503],accel_mss,speed_ms,0,blend_radius_m)
    |   movel([0.136781, -1.477052, -2.500928, -0.734409, 1.570796, 1.707577],accel_mss,speed_ms,0,blend_radius_m)
    |   movel([0.135944, -1.476068, -2.501764, -0.734557, 1.570796, 1.706740],accel_mss,speed_ms,0,blend_radius_m)
    |   movel([0.135624, -1.476478, -2.501415, -0.734495, 1.570796, 1.706421],accel_mss,speed_ms,0,blend_radius_m)
    |   movel([0.135418, -1.476911, -2.501048, -0.734430, 1.570796, 1.706214],accel_mss,speed_ms,0,blend_radius_m)
    |   movel([0.135301, -1.477824, -2.500271, -0.734294, 1.570796, 1.706097],accel_mss,speed_ms,0,blend_radius_m)
    |   movel([0.135502, -1.478767, -2.499468, -0.734155, 1.570796, 1.706298],accel_mss,speed_ms,0,blend_radius_m)
    |   movel([0.135937, -1.479701, -2.498670, -0.734018, 1.570796, 1.706733],accel_mss,speed_ms,0,blend_radius_m)
    |   movel([0.137146, -1.481406, -2.497211, -0.733772, 1.570796, 1.707942],accel_mss,speed_ms,0,blend_radius_m)
    |   movel([0.138235, -1.482636, -2.496156, -0.733597, 1.570796, 1.709031],accel_mss,speed_ms,0,blend_radius_m)
    |   movel([0.138569, -1.483138, -2.495724, -0.733527, 1.570796, 1.709366],accel_mss,speed_ms,0,blend_radius_m)
    |   movel([0.138615, -1.483435, -2.495469, -0.733485, 1.570796, 1.709411],accel_mss,speed_ms,0,blend_radius_m)
    |   movel([0.138508, -1.483765, -2.495185, -0.733439, 1.570796, 1.709305],accel_mss,speed_ms,0,blend_radius_m)
    |   movel([0.138244, -1.484095, -2.494901, -0.733393, 1.570796, 1.709040],accel_mss,speed_ms,0,blend_radius_m)
    |   movel([0.137948, -1.484275, -2.494745, -0.733368, 1.570796, 1.708744],accel_mss,speed_ms,0,blend_radius_m)
    |   movel([0.137318, -1.484345, -2.494686, -0.733359, 1.570796, 1.708115],accel_mss,speed_ms,0,blend_radius_m)
    |   movel([0.136454, -1.484350, -2.494681, -0.733358, 1.570796, 1.707250],accel_mss,speed_ms,0,blend_radius_m)
    |   movel([0.136239, -1.484493, -2.494558, -0.733338, 1.570796, 1.707035],accel_mss,speed_ms,0,blend_radius_m)
    |   movel([0.136059, -1.484791, -2.494301, -0.733297, 1.570796, 1.706856],accel_mss,speed_ms,0,blend_radius_m)
    |   movel([0.136003, -1.485128, -2.494010, -0.733251, 1.570796, 1.706800],accel_mss,speed_ms,0,blend_radius_m)
    |   movel([0.136163, -1.485852, -2.493385, -0.733152, 1.570796, 1.706959],accel_mss,speed_ms,0,blend_radius_m)
    |   movel([0.136787, -1.487054, -2.492345, -0.732990, 1.570796, 1.707583],accel_mss,speed_ms,0,blend_radius_m)
    |   movel([0.138315, -1.489476, -2.490244, -0.732670, 1.570796, 1.709111],accel_mss,speed_ms,0,blend_radius_m)
    |   movel([0.139902, -1.491849, -2.488175, -0.732365, 1.570796, 1.710698],accel_mss,speed_ms,0,blend_radius_m)
    |   movel([0.140129, -1.492382, -2.487709, -0.732298, 1.570796, 1.710925],accel_mss,speed_ms,0,blend_radius_m)
    |   movel([0.140207, -1.492984, -2.487182, -0.732223, 1.570796, 1.711003],accel_mss,speed_ms,0,blend_radius_m)
    |   movel([0.140047, -1.493584, -2.486657, -0.732148, 1.570796, 1.710844],accel_mss,speed_ms,0,blend_radius_m)
    |   movel([0.139855, -1.493859, -2.486416, -0.732114, 1.570796, 1.710651],accel_mss,speed_ms,0,blend_radius_m)
    |   movel([0.139253, -1.494278, -2.486048, -0.732063, 1.570796, 1.710049],accel_mss,speed_ms,0,blend_radius_m)
    |   movel([0.138942, -1.494367, -2.485971, -0.732052, 1.570796, 1.709738],accel_mss,speed_ms,0,blend_radius_m)
    |   movel([0.138342, -1.494337, -2.485996, -0.732055, 1.570796, 1.709138],accel_mss,speed_ms,0,blend_radius_m)
    |   movel([0.137803, -1.494114, -2.486193, -0.732083, 1.570796, 1.708599],accel_mss,speed_ms,0,blend_radius_m)
    |   movel([0.137358, -1.493785, -2.486481, -0.732123, 1.570796, 1.708154],accel_mss,speed_ms,0,blend_radius_m)
    |   movel([0.135058, -1.491567, -2.488421, -0.732401, 1.570796, 1.705854],accel_mss,speed_ms,0,blend_radius_m)
    |   movel([0.132918, -1.489209, -2.490475, -0.732704, 1.570796, 1.703714],accel_mss,speed_ms,0,blend_radius_m)
    |   movel([0.130949, -1.486712, -2.492642, -0.733036, 1.570796, 1.701746],accel_mss,speed_ms,0,blend_radius_m)
    |   movel([0.129157, -1.484079, -2.494915, -0.733395, 1.570796, 1.699953],accel_mss,speed_ms,0,blend_radius_m)
    |   movel([0.128568, -1.483052, -2.495799, -0.733539, 1.570796, 1.699364],accel_mss,speed_ms,0,blend_radius_m)
    |   movel([0.128197, -1.481908, -2.496781, -0.733700, 1.570796, 1.698993],accel_mss,speed_ms,0,blend_radius_m)
    |   movel([0.128149, -1.481157, -2.497425, -0.733808, 1.570796, 1.698945],accel_mss,speed_ms,0,blend_radius_m)
    |   movel([0.128212, -1.480370, -2.498098, -0.733921, 1.570796, 1.699008],accel_mss,speed_ms,0,blend_radius_m)
    |   movel([0.128521, -1.478745, -2.499487, -0.734158, 1.570796, 1.699317],accel_mss,speed_ms,0,blend_radius_m)
    |   movel([0.130258, -1.472804, -2.504525, -0.735059, 1.570796, 1.701055],accel_mss,speed_ms,0,blend_radius_m)
    |   movel([0.130584, -1.471144, -2.505924, -0.735321, 1.570796, 1.701380],accel_mss,speed_ms,0,blend_radius_m)
    |   movel([0.130664, -1.469682, -2.507152, -0.735555, 1.570796, 1.701461],accel_mss,speed_ms,0,blend_radius_m)
    |   movel([0.130585, -1.469067, -2.507667, -0.735655, 1.570796, 1.701381],accel_mss,speed_ms,0,blend_radius_m)
    |   movel([0.130405, -1.468553, -2.508097, -0.735738, 1.570796, 1.701201],accel_mss,speed_ms,0,blend_radius_m)
    |   movel([0.130115, -1.468156, -2.508429, -0.735803, 1.570796, 1.700911],accel_mss,speed_ms,0,blend_radius_m)
    |   movel([0.129704, -1.467894, -2.508649, -0.735846, 1.570796, 1.700500],accel_mss,speed_ms,0,blend_radius_m)
    |   movel([0.128816, -1.467662, -2.508842, -0.735884, 1.570796, 1.699612],accel_mss,speed_ms,0,blend_radius_m)
    |   movel([0.128423, -1.467505, -2.508974, -0.735910, 1.570796, 1.699220],accel_mss,speed_ms,0,blend_radius_m)
    |   movel([0.128171, -1.467225, -2.509208, -0.735956, 1.570796, 1.698967],accel_mss,speed_ms,0,blend_radius_m)
    |   movel([0.128179, -1.466606, -2.509724, -0.736059, 1.570796, 1.698975],accel_mss,speed_ms,0,blend_radius_m)
    |   movel([0.128477, -1.465914, -2.510301, -0.736174, 1.570796, 1.699274],accel_mss,speed_ms,0,blend_radius_m)
    |   movel([0.129531, -1.463700, -2.512141, -0.736548, 1.570796, 1.700328],accel_mss,speed_ms,0,blend_radius_m)
    |   movel([0.130435, -1.461494, -2.513967, -0.736928, 1.570796, 1.701231],accel_mss,speed_ms,0,blend_radius_m)
    |   movel([0.131207, -1.459289, -2.515784, -0.737316, 1.570796, 1.702003],accel_mss,speed_ms,0,blend_radius_m)
    |   movel([0.131868, -1.457083, -2.517594, -0.737711, 1.570796, 1.702664],accel_mss,speed_ms,0,blend_radius_m)
    |   movel([0.132952, -1.452659, -2.521204, -0.738527, 1.570796, 1.703749],accel_mss,speed_ms,0,blend_radius_m)
    |   movel([0.133860, -1.448187, -2.524821, -0.739381, 1.570796, 1.704656],accel_mss,speed_ms,0,blend_radius_m)
    |   speed_ms = 0.005
    |   movel([0.133860, -1.439913, -2.521119, -0.751357, 1.570796, 1.704656],accel_mss,speed_ms,0,blend_radius_m)
    |   speed_ms = 0.040
    |   movel([0.129330, -1.451283, -2.511982, -0.749125, 1.570796, 1.700127],accel_mss,speed_ms,0,blend_radius_m)
    |   speed_ms = 0.005
    |   movel([0.129330, -1.459468, -2.515637, -0.737284, 1.570796, 1.700127],accel_mss,speed_ms,0,blend_radius_m)
    |   speed_ms = 0.025
    |   movel([0.126610, -1.462183, -2.513397, -0.736809, 1.570796, 1.697407],accel_mss,speed_ms,0,blend_radius_m)
    |   movel([0.123791, -1.464805, -2.511224, -0.736361, 1.570796, 1.694587],accel_mss,speed_ms,0,blend_radius_m)
    |   movel([0.120879, -1.467331, -2.509119, -0.735939, 1.570796, 1.691675],accel_mss,speed_ms,0,blend_radius_m)
    |   movel([0.117884, -1.469751, -2.507094, -0.735544, 1.570796, 1.688680],accel_mss,speed_ms,0,blend_radius_m)
    |   movel([0.120109, -1.467090, -2.509320, -0.735979, 1.570796, 1.690905],accel_mss,speed_ms,0,blend_radius_m)
    |   movel([0.122141, -1.464340, -2.511609, -0.736439, 1.570796, 1.692938],accel_mss,speed_ms,0,blend_radius_m)
    |   movel([0.123966, -1.461520, -2.513945, -0.736924, 1.570796, 1.694762],accel_mss,speed_ms,0,blend_radius_m)
    |   movel([0.125570, -1.458647, -2.516312, -0.737430, 1.570796, 1.696366],accel_mss,speed_ms,0,blend_radius_m)
    |   movel([0.123268, -1.460861, -2.514489, -0.737039, 1.570796, 1.694064],accel_mss,speed_ms,0,blend_radius_m)
    |   movel([0.120894, -1.463001, -2.512720, -0.736668, 1.570796, 1.691690],accel_mss,speed_ms,0,blend_radius_m)
    |   movel([0.118447, -1.465068, -2.511005, -0.736316, 1.570796, 1.689244],accel_mss,speed_ms,0,blend_radius_m)
    |   movel([0.115936, -1.467052, -2.509352, -0.735985, 1.570796, 1.686733],accel_mss,speed_ms,0,blend_radius_m)
    |   movel([0.113105, -1.469202, -2.507554, -0.735633, 1.570796, 1.683901],accel_mss,speed_ms,0,blend_radius_m)
    |   movel([0.110401, -1.471457, -2.505661, -0.735272, 1.570796, 1.681198],accel_mss,speed_ms,0,blend_radius_m)
    |   movel([0.109168, -1.472687, -2.504625, -0.735078, 1.570796, 1.679965],accel_mss,speed_ms,0,blend_radius_m)
    |   movel([0.108074, -1.473989, -2.503525, -0.734875, 1.570796, 1.678871],accel_mss,speed_ms,0,blend_radius_m)
    |   movel([0.107185, -1.475341, -2.502380, -0.734668, 1.570796, 1.677982],accel_mss,speed_ms,0,blend_radius_m)
    |   movel([0.106556, -1.476720, -2.501210, -0.734459, 1.570796, 1.677352],accel_mss,speed_ms,0,blend_radius_m)
    |   movel([0.106935, -1.475038, -2.502637, -0.734714, 1.570796, 1.677731],accel_mss,speed_ms,0,blend_radius_m)
    |   movel([0.107478, -1.473291, -2.504114, -0.734983, 1.570796, 1.678274],accel_mss,speed_ms,0,blend_radius_m)
    |   movel([0.108174, -1.471503, -2.505621, -0.735264, 1.570796, 1.678970],accel_mss,speed_ms,0,blend_radius_m)
    |   movel([0.109010, -1.469695, -2.507140, -0.735553, 1.570796, 1.679807],accel_mss,speed_ms,0,blend_radius_m)
    |   movel([0.109974, -1.467891, -2.508651, -0.735847, 1.570796, 1.680770],accel_mss,speed_ms,0,blend_radius_m)
    |   movel([0.111053, -1.466112, -2.510136, -0.736141, 1.570796, 1.681850],accel_mss,speed_ms,0,blend_radius_m)
    |   movel([0.112236, -1.464382, -2.511574, -0.736432, 1.570796, 1.683032],accel_mss,speed_ms,0,blend_radius_m)
    |   movel([0.113506, -1.462726, -2.512948, -0.736715, 1.570796, 1.684303],accel_mss,speed_ms,0,blend_radius_m)
    |   movel([0.111148, -1.465240, -2.510862, -0.736287, 1.570796, 1.681944],accel_mss,speed_ms,0,blend_radius_m)
    |   movel([0.108940, -1.467810, -2.508719, -0.735860, 1.570796, 1.679736],accel_mss,speed_ms,0,blend_radius_m)
    |   movel([0.106873, -1.470424, -2.506528, -0.735436, 1.570796, 1.677669],accel_mss,speed_ms,0,blend_radius_m)
    |   movel([0.104936, -1.473073, -2.504299, -0.735017, 1.570796, 1.675732],accel_mss,speed_ms,0,blend_radius_m)
    |   movel([0.103122, -1.475740, -2.502042, -0.734607, 1.570796, 1.673918],accel_mss,speed_ms,0,blend_radius_m)
    |   movel([0.101418, -1.478416, -2.499767, -0.734206, 1.570796, 1.672214],accel_mss,speed_ms,0,blend_radius_m)
    |   movel([0.098300, -1.483746, -2.495201, -0.733442, 1.570796, 1.669096],accel_mss,speed_ms,0,blend_radius_m)
    |   movel([0.099115, -1.481886, -2.496800, -0.733703, 1.570796, 1.669911],accel_mss,speed_ms,0,blend_radius_m)
    |   movel([0.099701, -1.479887, -2.498512, -0.733991, 1.570796, 1.670497],accel_mss,speed_ms,0,blend_radius_m)
    |   movel([0.100679, -1.475992, -2.501828, -0.734569, 1.570796, 1.671475],accel_mss,speed_ms,0,blend_radius_m)
    |   movel([0.101284, -1.474259, -2.503297, -0.734834, 1.570796, 1.672081],accel_mss,speed_ms,0,blend_radius_m)
    |   movel([0.101969, -1.472701, -2.504612, -0.735076, 1.570796, 1.672765],accel_mss,speed_ms,0,blend_radius_m)
    |   movel([0.103697, -1.469504, -2.507301, -0.735584, 1.570796, 1.674493],accel_mss,speed_ms,0,blend_radius_m)
    |   movel([0.103298, -1.469937, -2.506938, -0.735514, 1.570796, 1.674094],accel_mss,speed_ms,0,blend_radius_m)
    |   movel([0.102596, -1.470462, -2.506497, -0.735430, 1.570796, 1.673392],accel_mss,speed_ms,0,blend_radius_m)
    |   movel([0.098578, -1.472860, -2.504478, -0.735051, 1.570796, 1.669375],accel_mss,speed_ms,0,blend_radius_m)
    |   movel([0.097137, -1.473796, -2.503688, -0.734905, 1.570796, 1.667933],accel_mss,speed_ms,0,blend_radius_m)
    |   movel([0.095576, -1.475228, -2.502477, -0.734685, 1.570796, 1.666372],accel_mss,speed_ms,0,blend_radius_m)
    |   movel([0.094153, -1.476803, -2.501140, -0.734446, 1.570796, 1.664949],accel_mss,speed_ms,0,blend_radius_m)
    |   movel([0.091623, -1.480067, -2.498357, -0.733965, 1.570796, 1.662419],accel_mss,speed_ms,0,blend_radius_m)
    |   movel([0.092560, -1.478289, -2.499875, -0.734225, 1.570796, 1.663356],accel_mss,speed_ms,0,blend_radius_m)
    |   movel([0.093335, -1.476490, -2.501406, -0.734494, 1.570796, 1.664131],accel_mss,speed_ms,0,blend_radius_m)
    |   movel([0.094831, -1.472870, -2.504470, -0.735049, 1.570796, 1.665628],accel_mss,speed_ms,0,blend_radius_m)
    |   movel([0.095802, -1.471000, -2.506045, -0.735344, 1.570796, 1.666598],accel_mss,speed_ms,0,blend_radius_m)
    |   movel([0.096940, -1.469133, -2.507612, -0.735644, 1.570796, 1.667736],accel_mss,speed_ms,0,blend_radius_m)
    |   movel([0.099590, -1.465408, -2.510722, -0.736259, 1.570796, 1.670387],accel_mss,speed_ms,0,blend_radius_m)
    |   movel([0.105374, -1.458093, -2.516767, -0.737529, 1.570796, 1.676170],accel_mss,speed_ms,0,blend_radius_m)
    |   movel([0.102945, -1.459280, -2.515791, -0.737317, 1.570796, 1.673741],accel_mss,speed_ms,0,blend_radius_m)
    |   movel([0.100569, -1.460608, -2.514698, -0.737083, 1.570796, 1.671365],accel_mss,speed_ms,0,blend_radius_m)
    |   movel([0.098254, -1.462062, -2.513497, -0.736830, 1.570796, 1.669051],accel_mss,speed_ms,0,blend_radius_m)
    |   movel([0.096018, -1.463634, -2.512196, -0.736560, 1.570796, 1.666815],accel_mss,speed_ms,0,blend_radius_m)
    |   movel([0.093877, -1.465311, -2.510803, -0.736275, 1.570796, 1.664673],accel_mss,speed_ms,0,blend_radius_m)
    |   movel([0.091839, -1.467084, -2.509325, -0.735980, 1.570796, 1.662635],accel_mss,speed_ms,0,blend_radius_m)
    |   movel([0.089918, -1.468941, -2.507773, -0.735675, 1.570796, 1.660714],accel_mss,speed_ms,0,blend_radius_m)
    |   movel([0.088128, -1.470872, -2.506152, -0.735364, 1.570796, 1.658924],accel_mss,speed_ms,0,blend_radius_m)
    |   movel([0.088591, -1.470264, -2.506663, -0.735462, 1.570796, 1.659388],accel_mss,speed_ms,0,blend_radius_m)
    |   movel([0.089010, -1.469568, -2.507247, -0.735574, 1.570796, 1.659806],accel_mss,speed_ms,0,blend_radius_m)
    |   movel([0.089748, -1.468019, -2.508544, -0.735826, 1.570796, 1.660544],accel_mss,speed_ms,0,blend_radius_m)
    |   movel([0.091069, -1.465035, -2.511033, -0.736322, 1.570796, 1.661865],accel_mss,speed_ms,0,blend_radius_m)
    |   movel([0.092511, -1.462509, -2.513127, -0.736752, 1.570796, 1.663307],accel_mss,speed_ms,0,blend_radius_m)
    |   movel([0.094073, -1.460009, -2.515192, -0.737189, 1.570796, 1.664869],accel_mss,speed_ms,0,blend_radius_m)
    |   movel([0.095749, -1.457534, -2.517226, -0.737630, 1.570796, 1.666545],accel_mss,speed_ms,0,blend_radius_m)
    |   movel([0.097530, -1.455082, -2.519231, -0.738076, 1.570796, 1.668326],accel_mss,speed_ms,0,blend_radius_m)
    |   movel([0.099411, -1.452649, -2.521212, -0.738528, 1.570796, 1.670208],accel_mss,speed_ms,0,blend_radius_m)
    |   movel([0.101389, -1.450236, -2.523167, -0.738986, 1.570796, 1.672185],accel_mss,speed_ms,0,blend_radius_m)
    |   movel([0.105602, -1.445450, -2.527019, -0.739920, 1.570796, 1.676399],accel_mss,speed_ms,0,blend_radius_m)
    |   movel([0.103770, -1.446818, -2.525922, -0.739649, 1.570796, 1.674566],accel_mss,speed_ms,0,blend_radius_m)
    |   movel([0.098045, -1.450583, -2.522887, -0.738920, 1.570796, 1.668841],accel_mss,speed_ms,0,blend_radius_m)
    |   movel([0.096170, -1.451893, -2.521825, -0.738671, 1.570796, 1.666966],accel_mss,speed_ms,0,blend_radius_m)
    |   movel([0.094379, -1.453303, -2.520680, -0.738406, 1.570796, 1.665176],accel_mss,speed_ms,0,blend_radius_m)
    |   movel([0.092747, -1.454825, -2.519440, -0.738124, 1.570796, 1.663543],accel_mss,speed_ms,0,blend_radius_m)
    |   movel([0.091340, -1.456474, -2.518094, -0.737822, 1.570796, 1.662136],accel_mss,speed_ms,0,blend_radius_m)
    |   movel([0.093177, -1.453658, -2.520392, -0.738340, 1.570796, 1.663973],accel_mss,speed_ms,0,blend_radius_m)
    |   movel([0.094978, -1.450714, -2.522780, -0.738895, 1.570796, 1.665775],accel_mss,speed_ms,0,blend_radius_m)
    |   movel([0.096894, -1.447801, -2.525131, -0.739457, 1.570796, 1.667691],accel_mss,speed_ms,0,blend_radius_m)
